(* CODESYS project BODAS-HelloWorld

Project tree, tasks and I/O mapping:
  BODAS_RC18_12_40 : BODAS_RC18-12_27-18_40, Bosch Rexroth AG, version 3.5.21.0
    application Application
      libraries: BODAS_RC18-12_27-18_40, 3.0.1 (Bosch Rexroth AG); BODAS_RC18-12_27-18_40-DST, 2.3.0 (Bosch Rexroth AG); BODAS_RC18-12_27-18_40-PR4, 2.3.0 (Bosch Rexroth AG); Util, 3.5.19.0 (System)
      task Os10msProc (cyclic, interval 10 ms, priority 1) calls MAIN_TASK_PRG
      00 Init/
        FunctionBlocks/
        program INIT_PRG [ST]: INIT_cfgInputs, INIT_cfgOutputs, INIT_initCAN, INIT_initNVM, INIT_initSys, INIT_initUDS
        Programs/
      01 MainTask/
        00 Startlock/
          FunctionBlocks/
          Programs/
        01 Inputs/
          FunctionBlocks/
          program PRG_Inputs [ST]: ACT_InitInputs
          Programs/
        02 Outputs/
          FunctionBlocks/
          program PRG_Outputs [ST]: ACT_HandleInhibit, ACT_InitOutputs
          program PRG_SafeOuts [ST]: ACT_InitSafeOutputs
          Programs/
        03 Communication/
          00 CAN/
            Function/
            FunctionBlocks/
            program PRG_CANIn [ST]
            program PRG_CANOut [ST]
            Programs/
          01 ISOBUSJ1939/
            FunctionBlocks/
            program PRG_ISOBUSJ1939 [ST]
            Programs/
          02 CANopen/
        04 Hydraulics/
          FunctionBlocks/
          Programs/
        05 Engine/
          FunctionBlocks/
          Programs/
        06 Drivetrain/
          FunctionBlocks/
          Programs/
        07 HMI/
          FunctionBlocks/
          Programs/
        10 Service/
          FunctionBlocks/
          program PRG_UDS [ST]: ACT_InitUDS
          Programs/
            program UDS_DefaultCallback [ST]
            function UDS_Diag_ChkLvl [ST]
            function UDS_ReadCallback [ST]
            program UDS_RoutineCallback [ST]
            function UDS_WriteCallback [ST]
        11 Parameters/
          FunctionBlocks/
          Functions/
            function FUNC_DbgMgrRisingEdgeDetn [ST]
          program PRG_DebugManager [ST]: ACT_InitDebugManager
          Programs/
            program PRG_NVMConfig [ST]
        20_Errors/
          FunctionBlocks/
          Functions/
          program PRG_ErrMemMgr [ST]: ACT_ClrDFESEntry, ACT_GetDFESEntry
          program PRG_HandleErrors [ST]: ACT_InitHandleErrors
          Programs/
      02 EasyConfig/
        DSM_easyConfig/
          GVL/
            global variables GVL_debounceMethod
          Structure/
            data type DFC_bds_NoDeb0x8000
            data type DFC_bds_NoDeb0x8001
            data type DFC_bds_NoDeb0x8002
            data type DFC_bds_NoDeb0x8003
            data type DFC_bds_NoDeb0x8004
            data type DFC_bds_NoDeb0x8005
            data type DFC_bds_NoDeb0x8006
            data type DFC_bds_NoDeb0x8007
            data type DFC_bds_NoDeb0x8008
            data type DFC_bds_NoDeb0x8009
            data type DFC_bds_NoDeb0x800a
            data type DFC_bds_NoDeb0x800b
            data type DFC_bds_NoDeb0x800c
            data type DFC_bds_NoDeb0x800d
            data type DFC_bds_NoDeb0x800e
            data type DFC_bds_NoDeb0x800f
            data type DFC_bds_NoDeb0x8010
            data type DFC_bds_NoDeb0x8011
            data type DFC_bds_NoDeb0x8012
            data type DFC_bds_NoDeb0x8013
            data type DFC_bds_NoDeb0x8014
            data type DFC_bds_NoDeb0x8015
            data type DFC_bds_NoDeb0x8016
            data type DFC_bds_NoDeb0x8017
            data type DFC_bds_NoDeb0x8018
            data type DFC_bds_NoDeb0x8019
            data type DFC_bds_NoDeb0x801a
            data type DFC_bds_NoDeb0x801b
            data type DFC_bds_NoDeb0x801c
            data type DFC_bds_NoDeb0x801d
            data type DFC_bds_NoDeb0x801e
            data type DFC_bds_NoDeb0x801f
            data type DFC_bds_NoDeb0x8020
            data type DFC_bds_NoDeb0x8021
            data type DFC_bds_NoDeb0x8022
            data type DFC_bds_NoDeb0x8023
            data type DFC_bds_NoDeb0x8024
            data type DFC_bds_NoDeb0x8025
            data type DFC_bds_NoDeb0x8026
            data type DFC_bds_NoDeb0x8027
            data type DFC_bds_NoDeb0x8028
            data type DFC_bds_NoDeb0x8029
            data type DFC_bds_NoDeb0x802a
            data type DFC_bds_NoDeb0x802b
            data type DFC_bds_NoDeb0x802c
            data type DFC_bds_NoDeb0x802d
            data type DFC_bds_NoDeb0x802e
            data type DFC_bds_NoDeb0x802f
            data type DFC_bds_NoDeb0x8030
            data type DFC_bds_NoDeb0x8031
            data type DFC_bds_NoDeb0x8032
            data type DFC_bds_NoDeb0x8033
            data type DFC_bds_NoDeb0x8034
            data type DFC_bds_NoDeb0x8035
            data type DFC_bds_NoDeb0x8036
            data type DFC_bds_NoDeb0x8037
            data type DFC_bds_NoDeb0x8038
            data type DFC_bds_NoDeb0x8039
            data type DFC_bds_NoDeb0x803a
            data type DFC_bds_NoDeb0x803b
            data type DFC_bds_NoDeb0x803c
            data type DFC_bds_NoDeb0x803d
            data type DFC_bds_NoDeb0x803e
            data type DFC_bds_NoDeb0x803f
            data type DFC_bds_NoDeb0x8040
            data type DFC_bds_NoDeb0x8041
            data type DFC_bds_NoDeb0x8042
            data type DFC_bds_NoDeb0x8043
            data type DFC_bds_NoDeb0x8044
            data type DFC_bds_NoDeb0x8045
            data type DFC_bds_NoDeb0x8046
            data type DFC_bds_NoDeb0x8047
            data type DFC_bds_NoDeb0x8048
            data type DFC_bds_NoDeb0x8049
            data type DFC_bds_NoDeb0x804a
            data type DFC_bds_NoDeb0x804b
            data type DFC_bds_NoDeb0x804c
            data type DFC_bds_NoDeb0x804d
            data type DFC_bds_NoDeb0x804e
            data type DFC_bds_NoDeb0x804f
            data type DFC_bds_NoDeb0x8050
            data type DFC_bds_NoDeb0x8051
            data type DFC_bds_NoDeb0x8052
            data type DFC_bds_NoDeb0x8053
            data type DFC_bds_NoDeb0x8054
            data type DFC_bds_NoDeb0x8055
            data type DFC_bds_NoDeb0x8056
            data type DFC_bds_NoDeb0x8057
            data type DFC_bds_NoDeb0x8058
            data type DFC_bds_NoDeb0x8059
            data type DFC_bds_NoDeb0x805a
            data type DFC_bds_NoDeb0x805b
            data type DFC_bds_NoDeb0x805c
            data type DFC_bds_NoDeb0x805d
            data type DFC_bds_NoDeb0x805e
            data type DFC_bds_NoDeb0x805f
            data type DFC_bds_NoDeb0x8060
            data type DFC_bds_NoDeb0x8061
            data type DFC_bds_NoDeb0x8062
            data type DFC_bds_NoDeb0x8063
            data type DFC_bds_NoDeb0x8064
            data type DFC_bds_NoDeb0x8065
            data type DFC_bds_NoDeb0x8066
            data type DFC_bds_NoDeb0x8067
            data type DFC_bds_NoDeb0x8068
            data type DFC_bds_NoDeb0x8069
            data type DFC_bds_NoDeb0x806a
            data type DFC_bds_NoDeb0x806b
            data type DFC_bds_NoDeb0x806c
            data type DFC_bds_NoDeb0x806d
            data type DFC_bds_NoDeb0x806e
            data type DFC_bds_NoDeb0x806f
            data type DFC_bds_NoDeb0x8070
            data type DFC_bds_NoDeb0x8071
            data type DFC_bds_NoDeb0x8072
            data type DFC_bds_NoDeb0x8073
            data type DFC_bds_NoDeb0x8074
            data type DFC_bds_NoDeb0x8075
            data type DFC_bds_NoDeb0x8076
            data type DFC_bds_NoDeb0x8077
            data type DFC_bds_NoDeb0x8078
            data type DFC_bds_NoDeb0x8079
            data type DFC_bds_NoDeb0x807a
            data type DFC_bds_NoDeb0x807b
            data type DFC_bds_NoDeb0x807c
            data type DFC_bds_NoDeb0x807d
            data type DFC_bds_NoDeb0x807e
            data type DFC_bds_NoDeb0x807f
            data type DFC_bds_NoDeb0x8080
            data type DFC_bds_NoDeb0x8081
            data type DFC_bds_NoDeb0x8082
            data type DFC_bds_NoDeb0x8083
            data type DFC_bds_NoDeb0x8084
            data type DFC_bds_NoDeb0x8085
            data type DFC_bds_NoDeb0x8086
            data type DFC_bds_NoDeb0x8087
            data type DFC_bds_NoDeb0x8088
            data type DFC_bds_NoDeb0x8089
            data type DFC_bds_NoDeb0x808a
            data type DFC_bds_NoDeb0x808b
            data type DFC_bds_NoDeb0x808c
            data type DFC_bds_NoDeb0x808d
            data type DFC_bds_NoDeb0x808e
            data type DFC_bds_NoDeb0x808f
            data type DFC_bds_NoDeb0x8090
            data type DFC_bds_NoDeb0x8091
            data type DFC_bds_NoDeb0x8092
            data type DFC_bds_NoDeb0x8093
            data type DFC_bds_NoDeb0x8094
            data type DFC_bds_NoDeb0x8095
            data type DFC_bds_NoDeb0x8096
            data type DFC_bds_NoDeb0x8097
            data type DFC_bds_NoDeb0x8098
            data type DFC_bds_NoDeb0x8099
            data type DFC_bds_NoDeb0x809a
            data type DFC_bds_NoDeb0x809b
            data type DFC_bds_NoDeb0x809c
            data type DFC_bds_NoDeb0x809d
            data type DFC_bds_NoDeb0x809e
            data type DFC_bds_NoDeb0x809f
            data type DFC_bds_NoDeb0x80a0
            data type DFC_bds_NoDeb0x80a1
            data type DFC_bds_NoDeb0x80a2
            data type DFC_bds_NoDeb0x80a3
            data type DFC_bds_NoDeb0x80a4
            data type DFC_bds_NoDeb0x80a5
            data type DFC_bds_NoDeb0x80a6
            data type DFC_bds_NoDeb0x80a7
            data type DFC_bds_NoDeb0x80a8
            data type DFC_bds_NoDeb0x80a9
            data type DFC_bds_NoDeb0x80aa
            data type DFC_bds_NoDeb0x80ab
            data type DFC_bds_NoDeb0x80ac
            data type DFC_bds_NoDeb0x80ad
            data type DFC_bds_NoDeb0x80ae
            data type DFC_bds_NoDeb0x80af
            data type DFC_bds_NoDeb0x80b0
            data type DFC_bds_NoDeb0x80b1
            data type DFC_bds_NoDeb0x80b2
            data type DFC_bds_NoDeb0x80b3
            data type DFC_bds_NoDeb0x80b4
            data type DFC_bds_NoDeb0x80b5
            data type DFC_bds_NoDeb0x80b6
            data type DFC_bds_NoDeb0x80b7
            data type DFC_bds_NoDeb0x80b8
            data type DFC_bds_NoDeb0x80b9
            data type DFC_bds_NoDeb0x80ba
            data type DFC_bds_NoDeb0x80bb
            data type DFC_bds_NoDeb0x80bc
            data type DFC_bds_NoDeb0x80bd
            data type DFC_bds_NoDeb0x80be
            data type DFC_bds_NoDeb0x80bf
            data type DFC_bds_NoDeb0x80c0
            data type DFC_bds_NoDeb0x80c1
            data type DFC_bds_NoDeb0x80c2
            data type DFC_bds_NoDeb0x80c3
            data type DFC_bds_NoDeb0x80c4
            data type DFC_bds_NoDeb0x80c5
            data type DFC_bds_NoDeb0x80c6
            data type DFC_bds_NoDeb0x80c7
            data type DFC_bds_NoDeb0x80c8
            data type DFC_bds_NoDeb0x80c9
            data type DFC_bds_NoDeb0x80ca
            data type DFC_bds_NoDeb0x80cb
            data type DFC_bds_NoDeb0x80cc
            data type DFC_bds_NoDeb0x80cd
            data type DFC_bds_NoDeb0x80ce
            data type DFC_bds_NoDeb0x80cf
            data type DFC_bds_NoDeb0x80d0
            data type DFC_bds_NoDeb0x80d1
            data type DFC_bds_NoDeb0x80d2
            data type DFC_bds_NoDeb0x80d3
            data type DFC_bds_NoDeb0x80d4
            data type DFC_bds_NoDeb0x80d5
            data type DFC_bds_NoDeb0x80d6
            data type DFC_bds_NoDeb0x80d7
            data type DFC_bds_NoDeb0x80d8
            data type DFC_bds_NoDeb0x80d9
            data type DFC_bds_NoDeb0x80da
            data type DFC_bds_NoDeb0x80db
            data type DFC_bds_NoDeb0x80dc
            data type DFC_bds_NoDeb0x80dd
            data type DFC_bds_NoDeb0x80de
            data type DFC_bds_NoDeb0x80df
            data type DFC_bds_NoDeb0x80e0
            data type DFC_bds_NoDeb0x80e1
            data type DFC_bds_NoDeb0x80e2
            data type DFC_bds_NoDeb0x80e3
            data type DFC_bds_NoDeb0x80e4
            data type DFC_bds_NoDeb0x80e5
            data type DFC_bds_NoDeb0x80e6
            data type DFC_bds_NoDeb0x80e7
            data type DFC_bds_NoDeb0x80e8
            data type DFC_bds_NoDeb0x80e9
            data type DFC_bds_NoDeb0x80ea
            data type DFC_bds_NoDeb0x80eb
            data type DFC_bds_NoDeb0x80ec
            data type DFC_bds_NoDeb0x80ed
            data type DFC_bds_NoDeb0x80ee
            data type DFC_bds_NoDeb0x80ef
            data type DFC_bds_NoDeb0x80f0
            data type DFC_bds_NoDeb0x80f1
            data type DFC_bds_NoDeb0x80f2
            data type DFC_bds_NoDeb0x80f3
            data type DFC_bds_NoDeb0x80f4
            data type DFC_bds_NoDeb0x80f5
            data type DFC_bds_NoDeb0x80f6
            data type DFC_bds_NoDeb0x80f7
            data type DFC_bds_NoDeb0x80f8
            data type DFC_bds_NoDeb0x80f9
            data type DFC_bds_NoDeb0x80fa
            data type DFC_bds_NoDeb0x80fb
            data type DFC_bds_NoDeb0x80fc
            data type DFC_bds_NoDeb0x80fd
            data type DFC_bds_NoDeb0x80fe
            data type DFC_bds_NoDeb0x80ff
            data type DFC_bds_NoDeb0x8100
            data type DFC_bds_NoDeb0x8101
            data type DFC_bds_NoDeb0x8102
            data type DFC_bds_NoDeb0x8103
            data type DFC_bds_NoDeb0x8104
            data type DFC_bds_NoDeb0x8105
            data type DFC_bds_NoDeb0x8106
            data type DFC_bds_NoDeb0x8107
            data type DFC_bds_NoDeb0x8108
            data type DFC_bds_NoDeb0x8109
            data type DFC_bds_NoDeb0x810a
            data type DFC_bds_NoDeb0x810b
            data type DFC_bds_NoDeb0x810c
            data type DFC_bds_NoDeb0x810d
            data type DFC_bds_NoDeb0x810e
            data type DFC_bds_NoDeb0x810f
            data type DFC_bds_NoDeb0x8110
            data type DFC_bds_NoDeb0x8111
            data type DFC_bds_NoDeb0x8112
            data type DFC_bds_NoDeb0x8113
            data type DFC_bds_NoDeb0x8114
            data type DFC_bds_NoDeb0x8115
            data type DFC_bds_NoDeb0x8116
            data type DFC_bds_NoDeb0x8117
            data type DFC_bds_NoDeb0x8118
            data type DFC_bds_NoDeb0x8119
            data type DFC_bds_NoDeb0x811a
            data type DFC_bds_NoDeb0x811b
            data type DFC_bds_NoDeb0x811c
            data type DFC_bds_NoDeb0x811d
            data type DFC_bds_NoDeb0x811e
            data type DFC_bds_NoDeb0x811f
            data type DFC_bds_NoDeb0x8120
            data type DFC_bds_NoDeb0x8121
            data type DFC_bds_NoDeb0x8122
            data type DFC_bds_NoDeb0x8123
            data type DFC_bds_NoDeb0x8124
            data type DFC_bds_NoDeb0x8125
            data type DFC_bds_NoDeb0x8126
            data type DFC_bds_NoDeb0x8127
            data type DFC_bds_NoDeb0x8128
            data type DFC_bds_NoDeb0x8129
            data type DFC_bds_NoDeb0x812a
            data type DFC_bds_NoDeb0x8C01
            data type DFC_bds_NoDeb0x8C02
            data type DFC_bds_NoDeb0x8C03
            data type DFC_bds_TiInRow0x8B01
            data type DFC_bds_TiInRow0x8B02
            data type DFC_bds_TiInRow0x8B03
            data type DFC_bds_TiUpDwn0x8A01
            data type DFC_bds_TiUpDwn0x8A02
            data type DFC_bds_TiUpDwn0x8A03
            data type DFC_CAN_E_TIMEOUT
            data type DFC_CANSM_E_BUS_OFF_NETWORK_0
            data type DFC_CANSM_E_BUS_OFF_NETWORK_1
            data type DFC_CANSM_E_BUS_OFF_NETWORK_2
            data type DFC_CANSM_E_BUS_OFF_NETWORK_3
            data type DFC_CANTRCV_E_NO_TRCV_CONTROL_0
            data type DFC_Com_numWhlIncFrtLeft
            data type DFC_Com_stWhlSensRrRht
            data type DFC_Com_trqClthTCSDCSDes
            data type DFC_Com_vWhlRrL
            data type DFC_ComChksACC_06
            data type DFC_ComChksBMS_01
            data type DFC_ComChksESP_02
            data type DFC_ComChksESP_05
            data type DFC_ComChksESP_07
            data type DFC_ComChksESP_10
            data type DFC_ComChksESP_19
            data type DFC_ComChksESP_20
            data type DFC_ComChksESP_21
            data type DFC_ComChksKlemmen_Status_01
            data type DFC_ComCntACC_06
            data type DFC_ComCntBMS_01
            data type DFC_ComCntESP_02
            data type DFC_ComCntESP_05
            data type DFC_ComCntESP_07
            data type DFC_ComCntESP_10
            data type DFC_ComCntESP_19
            data type DFC_ComCntESP_20
            data type DFC_ComCntESP_21
            data type DFC_ComCntKlemmen_Status_01
            data type DFC_ComDlcACC_06
            data type DFC_ComDlcESP_02
            data type DFC_ComDlcESP_05
            data type DFC_ComDlcESP_07
            data type DFC_ComDlcESP_10
            data type DFC_ComDlcESP_19
            data type DFC_ComDlcESP_20
            data type DFC_ComDlcESP_21
            data type DFC_COMM_E_NET_START_IND_CHANNEL_0
            data type DFC_COMM_E_NET_START_IND_CHANNEL_1
            data type DFC_COMM_E_NET_START_IND_CHANNEL_2
            data type DFC_COMM_E_NET_START_IND_CHANNEL_3
            data type DFC_COMM_E_NET_START_IND_CHANNEL_4
            data type DFC_COMM_E_NET_START_IND_CHANNEL_5
            data type DFC_ComTOutACC_06
            data type DFC_ComTOutESP_02
            data type DFC_ComTOutESP_05
            data type DFC_ComTOutESP_07
            data type DFC_ComTOutESP_10
            data type DFC_ComTOutESP_19
            data type DFC_ComTOutESP_20
            data type DFC_ComTOutESP_21
            data type DFC_DevLibBattUHi
            data type DFC_DevLibBattULo
            data type DFC_DSMDummy
            data type DFC_LIN_E_TIMEOUT
            data type DFC_MoCSOPICO
            data type DFC_MoFVarPostBldSel
            data type DFC_MoSysCtrlReIni
            data type DFC_MOXEMM_SMU_ALM0_0
            data type DFC_MOXEMM_SMU_ALM0_10
            data type DFC_MOXEMM_SMU_ALM0_11
            data type DFC_MOXEMM_SMU_ALM0_13
            data type DFC_MOXEMM_SMU_ALM0_14
            data type DFC_MOXEMM_SMU_ALM0_1
            data type DFC_MOXEMM_SMU_ALM0_22
            data type DFC_MOXEMM_SMU_ALM0_23
            data type DFC_MOXEMM_SMU_ALM0_2
            data type DFC_MOXEMM_SMU_ALM0_4
            data type DFC_MOXEMM_SMU_ALM0_5
            data type DFC_MOXEMM_SMU_ALM0_7
            data type DFC_MOXEMM_SMU_ALM0_8
            data type DFC_MOXEMM_SMU_ALM10_16
            data type DFC_MOXEMM_SMU_ALM10_17
            data type DFC_MOXEMM_SMU_ALM10_21
            data type DFC_MOXEMM_SMU_ALM11_0
            data type DFC_MOXEMM_SMU_ALM11_1
            data type DFC_MOXEMM_SMU_ALM11_2
            data type DFC_MOXEMM_SMU_ALM11_3
            data type DFC_MOXEMM_SMU_ALM11_4
            data type DFC_MOXEMM_SMU_ALM11_5
            data type DFC_MOXEMM_SMU_ALM11_8
            data type DFC_MOXEMM_SMU_ALM11_9
            data type DFC_MOXEMM_SMU_ALM1_0
            data type DFC_MOXEMM_SMU_ALM1_10
            data type DFC_MOXEMM_SMU_ALM1_11
            data type DFC_MOXEMM_SMU_ALM1_13
            data type DFC_MOXEMM_SMU_ALM1_14
            data type DFC_MOXEMM_SMU_ALM1_1
            data type DFC_MOXEMM_SMU_ALM1_22
            data type DFC_MOXEMM_SMU_ALM1_23
            data type DFC_MOXEMM_SMU_ALM1_2
            data type DFC_MOXEMM_SMU_ALM1_4
            data type DFC_MOXEMM_SMU_ALM1_5
            data type DFC_MOXEMM_SMU_ALM1_7
            data type DFC_MOXEMM_SMU_ALM1_8
            data type DFC_MOXEMM_SMU_ALM21_0
            data type DFC_MOXEMM_SMU_ALM21_16
            data type DFC_MOXEMM_SMU_ALM21_3
            data type DFC_MOXEMM_SMU_ALM2_10
            data type DFC_MOXEMM_SMU_ALM2_11
            data type DFC_MOXEMM_SMU_ALM2_13
            data type DFC_MOXEMM_SMU_ALM2_14
            data type DFC_MOXEMM_SMU_ALM2_1
            data type DFC_MOXEMM_SMU_ALM2_22
            data type DFC_MOXEMM_SMU_ALM2_23
            data type DFC_MOXEMM_SMU_ALM2_2
            data type DFC_MOXEMM_SMU_ALM2_4
            data type DFC_MOXEMM_SMU_ALM2_5
            data type DFC_MOXEMM_SMU_ALM2_7
            data type DFC_MOXEMM_SMU_ALM2_8
            data type DFC_MOXEMM_SMU_ALM3_10
            data type DFC_MOXEMM_SMU_ALM3_11
            data type DFC_MOXEMM_SMU_ALM3_13
            data type DFC_MOXEMM_SMU_ALM3_14
            data type DFC_MOXEMM_SMU_ALM3_1
            data type DFC_MOXEMM_SMU_ALM3_22
            data type DFC_MOXEMM_SMU_ALM3_23
            data type DFC_MOXEMM_SMU_ALM3_2
            data type DFC_MOXEMM_SMU_ALM3_4
            data type DFC_MOXEMM_SMU_ALM3_5
            data type DFC_MOXEMM_SMU_ALM3_7
            data type DFC_MOXEMM_SMU_ALM3_8
            data type DFC_MOXEMM_SMU_ALM6_0
            data type DFC_MOXEMM_SMU_ALM6_11
            data type DFC_MOXEMM_SMU_ALM6_12
            data type DFC_MOXEMM_SMU_ALM6_14
            data type DFC_MOXEMM_SMU_ALM6_15
            data type DFC_MOXEMM_SMU_ALM6_17
            data type DFC_MOXEMM_SMU_ALM6_18
            data type DFC_MOXEMM_SMU_ALM6_20
            data type DFC_MOXEMM_SMU_ALM6_21
            data type DFC_MOXEMM_SMU_ALM6_25
            data type DFC_MOXEMM_SMU_ALM6_2
            data type DFC_MOXEMM_SMU_ALM6_4
            data type DFC_MOXEMM_SMU_ALM6_5
            data type DFC_MOXEMM_SMU_ALM6_7
            data type DFC_MOXEMM_SMU_ALM6_8
            data type DFC_MOXEMM_SMU_ALM7_12
            data type DFC_MOXEMM_SMU_ALM7_13
            data type DFC_MOXEMM_SMU_ALM7_14
            data type DFC_MOXEMM_SMU_ALM7_15
            data type DFC_MOXEMM_SMU_ALM7_16
            data type DFC_MOXEMM_SMU_ALM7_17
            data type DFC_MOXEMM_SMU_ALM7_1
            data type DFC_MOXEMM_SMU_ALM7_20
            data type DFC_MOXEMM_SMU_ALM7_25
            data type DFC_MOXEMM_SMU_ALM7_26
            data type DFC_MOXEMM_SMU_ALM7_28
            data type DFC_MOXEMM_SMU_ALM7_29
            data type DFC_MOXEMM_SMU_ALM7_2
            data type DFC_MOXEMM_SMU_ALM7_30
            data type DFC_MOXEMM_SMU_ALM7_31
            data type DFC_MOXEMM_SMU_ALM8_0
            data type DFC_MOXEMM_SMU_ALM8_10
            data type DFC_MOXEMM_SMU_ALM8_11
            data type DFC_MOXEMM_SMU_ALM8_12
            data type DFC_MOXEMM_SMU_ALM8_13
            data type DFC_MOXEMM_SMU_ALM8_16
            data type DFC_MOXEMM_SMU_ALM8_18
            data type DFC_MOXEMM_SMU_ALM8_1
            data type DFC_MOXEMM_SMU_ALM8_2
            data type DFC_MOXEMM_SMU_ALM8_30
            data type DFC_MOXEMM_SMU_ALM8_31
            data type DFC_MOXEMM_SMU_ALM8_3
            data type DFC_MOXEMM_SMU_ALM8_4
            data type DFC_MOXEMM_SMU_ALM9_0
            data type DFC_MOXEMM_SMU_ALM9_15
            data type DFC_MOXEMM_SMU_ALM9_1
            data type DFC_MOXEMM_SMU_ALM9_3
            data type DFC_MoXEMMHwLTLBIST
            data type DFC_MoXEMMHwLTMBIST
            data type DFC_MoXEMMHwLTMCUFW
            data type DFC_MoXEMMHwLTMonBIST
            data type DFC_MoXEMMHwLTRegMonTest
            data type DFC_MoXEMMHwLTStbySMUAlvTest
        easyConfig_import/
          BDL/
          bds_in_ec/
          bds_in_legacy_ec/
          bds_out_ec/
          bds_sent_ec/
          bds_sysIo_ec/
          bds_sysPb_ec/
        Lin_CanSignals_easyConfig/
          global variables GVL_linCanSignals_easyConfig
      03 PrivateLibrary/
        DataTypes/
          DebugManager/
          ErrMemMgr/
          ISOBUSJ1939/
          MainTask/
      global variables GlobalVariables
      program MAIN_TASK_PRG [ST]: CAN_OUT, ERRORS, INIT, INPUTS, OUTPUTS, POSTRUN, READ_PARAMETERS, RUN, STARTLOCK
*)

// BODAS_RC18_12_40/Application/02 EasyConfig/DSM_easyConfig/Structure/DFC_bds_NoDeb0x8000
{attribute 'external_name' := 'cmp_rts_DFC_bds_NoDeb0x8000'}
TYPE DFC_bds_NoDeb0x8000 : STRUCT
        DTC            : UDINT := 16#800000;
        DFCid          : UINT  := 721;
        debounceMethod : USINT := NO_DEBOUNCE;
    END_STRUCT
END_TYPE

// BODAS_RC18_12_40/Application/02 EasyConfig/DSM_easyConfig/Structure/DFC_bds_NoDeb0x8001
{attribute 'external_name' := 'cmp_rts_DFC_bds_NoDeb0x8001'}
TYPE DFC_bds_NoDeb0x8001 : STRUCT
        DTC            : UDINT := 16#800100;
        DFCid          : UINT  := 722;
        debounceMethod : USINT := NO_DEBOUNCE;
    END_STRUCT
END_TYPE

// BODAS_RC18_12_40/Application/02 EasyConfig/DSM_easyConfig/Structure/DFC_bds_NoDeb0x8002
{attribute 'external_name' := 'cmp_rts_DFC_bds_NoDeb0x8002'}
TYPE DFC_bds_NoDeb0x8002 : STRUCT
        DTC            : UDINT := 16#800200;
        DFCid          : UINT  := 723;
        debounceMethod : USINT := NO_DEBOUNCE;
    END_STRUCT
END_TYPE

// BODAS_RC18_12_40/Application/02 EasyConfig/DSM_easyConfig/Structure/DFC_bds_NoDeb0x8003
{attribute 'external_name' := 'cmp_rts_DFC_bds_NoDeb0x8003'}
TYPE DFC_bds_NoDeb0x8003 : STRUCT
        DTC            : UDINT := 16#800300;
        DFCid          : UINT  := 724;
        debounceMethod : USINT := NO_DEBOUNCE;
    END_STRUCT
END_TYPE

// BODAS_RC18_12_40/Application/02 EasyConfig/DSM_easyConfig/Structure/DFC_bds_NoDeb0x8004
{attribute 'external_name' := 'cmp_rts_DFC_bds_NoDeb0x8004'}
TYPE DFC_bds_NoDeb0x8004 : STRUCT
        DTC            : UDINT := 16#800400;
        DFCid          : UINT  := 725;
        debounceMethod : USINT := NO_DEBOUNCE;
    END_STRUCT
END_TYPE

// BODAS_RC18_12_40/Application/02 EasyConfig/DSM_easyConfig/Structure/DFC_bds_NoDeb0x8005
{attribute 'external_name' := 'cmp_rts_DFC_bds_NoDeb0x8005'}
TYPE DFC_bds_NoDeb0x8005 :
STRUCT
	DTC: UDINT := 16#800500;
	DFCid: UINT := 726;
	debounceMethod: USINT := NO_DEBOUNCE;
END_STRUCT
END_TYPE

// BODAS_RC18_12_40/Application/02 EasyConfig/DSM_easyConfig/Structure/DFC_bds_NoDeb0x8006
{attribute 'external_name' := 'cmp_rts_DFC_bds_NoDeb0x8006'}
TYPE DFC_bds_NoDeb0x8006 : STRUCT
        DTC            : UDINT := 16#800600;
        DFCid          : UINT  := 727;
        debounceMethod : USINT := NO_DEBOUNCE;
    END_STRUCT
END_TYPE

// BODAS_RC18_12_40/Application/02 EasyConfig/DSM_easyConfig/Structure/DFC_bds_NoDeb0x8007
{attribute 'external_name' := 'cmp_rts_DFC_bds_NoDeb0x8007'}
TYPE DFC_bds_NoDeb0x8007 : STRUCT
        DTC            : UDINT := 16#800700;
        DFCid          : UINT  := 728;
        debounceMethod : USINT := NO_DEBOUNCE;
    END_STRUCT
END_TYPE

// BODAS_RC18_12_40/Application/02 EasyConfig/DSM_easyConfig/Structure/DFC_bds_NoDeb0x8008
{attribute 'external_name' := 'cmp_rts_DFC_bds_NoDeb0x8008'}
TYPE DFC_bds_NoDeb0x8008 : STRUCT
        DTC            : UDINT := 16#800800;
        DFCid          : UINT  := 729;
        debounceMethod : USINT := NO_DEBOUNCE;
    END_STRUCT
END_TYPE

// BODAS_RC18_12_40/Application/02 EasyConfig/DSM_easyConfig/Structure/DFC_bds_NoDeb0x8009
{attribute 'external_name' := 'cmp_rts_DFC_bds_NoDeb0x8009'}
TYPE DFC_bds_NoDeb0x8009 :
STRUCT
	DTC: UDINT := 16#800900;
	DFCid: UINT := 730;
	debounceMethod: USINT := NO_DEBOUNCE;
END_STRUCT
END_TYPE

// BODAS_RC18_12_40/Application/02 EasyConfig/DSM_easyConfig/Structure/DFC_bds_NoDeb0x800a
{attribute 'external_name' := 'cmp_rts_DFC_bds_NoDeb0x800a'}
TYPE DFC_bds_NoDeb0x800a : STRUCT
        DTC            : UDINT := 16#800A00;
        DFCid          : UINT  := 731;
        debounceMethod : USINT := NO_DEBOUNCE;
    END_STRUCT
END_TYPE

// BODAS_RC18_12_40/Application/02 EasyConfig/DSM_easyConfig/Structure/DFC_bds_NoDeb0x800b
{attribute 'external_name' := 'cmp_rts_DFC_bds_NoDeb0x800b'}
TYPE DFC_bds_NoDeb0x800b : STRUCT
        DTC            : UDINT := 16#800B00;
        DFCid          : UINT  := 732;
        debounceMethod : USINT := NO_DEBOUNCE;
    END_STRUCT
END_TYPE

// BODAS_RC18_12_40/Application/02 EasyConfig/DSM_easyConfig/Structure/DFC_bds_NoDeb0x800c
{attribute 'external_name' := 'cmp_rts_DFC_bds_NoDeb0x800c'}
TYPE DFC_bds_NoDeb0x800c :
STRUCT
	DTC: UDINT := 16#800C00;
	DFCid: UINT := 733;
	debounceMethod: USINT := NO_DEBOUNCE;
END_STRUCT
END_TYPE

// BODAS_RC18_12_40/Application/02 EasyConfig/DSM_easyConfig/Structure/DFC_bds_NoDeb0x800d
{attribute 'external_name' := 'cmp_rts_DFC_bds_NoDeb0x800d'}
TYPE DFC_bds_NoDeb0x800d : STRUCT
        DTC            : UDINT := 16#800D00;
        DFCid          : UINT  := 734;
        debounceMethod : USINT := NO_DEBOUNCE;
    END_STRUCT
END_TYPE

// BODAS_RC18_12_40/Application/02 EasyConfig/DSM_easyConfig/Structure/DFC_bds_NoDeb0x800e
{attribute 'external_name' := 'cmp_rts_DFC_bds_NoDeb0x800e'}
TYPE DFC_bds_NoDeb0x800e :
STRUCT
	DTC: UDINT := 16#800E00;
	DFCid: UINT := 735;
	debounceMethod: USINT := NO_DEBOUNCE;
END_STRUCT
END_TYPE

// BODAS_RC18_12_40/Application/02 EasyConfig/DSM_easyConfig/Structure/DFC_bds_NoDeb0x800f
{attribute 'external_name' := 'cmp_rts_DFC_bds_NoDeb0x800f'}
TYPE DFC_bds_NoDeb0x800f : STRUCT
        DTC            : UDINT := 16#800F00;
        DFCid          : UINT  := 736;
        debounceMethod : USINT := NO_DEBOUNCE;
    END_STRUCT
END_TYPE

// BODAS_RC18_12_40/Application/02 EasyConfig/DSM_easyConfig/Structure/DFC_bds_NoDeb0x8010
{attribute 'external_name' := 'cmp_rts_DFC_bds_NoDeb0x8010'}
TYPE DFC_bds_NoDeb0x8010 : STRUCT
        DTC            : UDINT := 16#801000;
        DFCid          : UINT  := 737;
        debounceMethod : USINT := NO_DEBOUNCE;
    END_STRUCT
END_TYPE

// BODAS_RC18_12_40/Application/02 EasyConfig/DSM_easyConfig/Structure/DFC_bds_NoDeb0x8011
{attribute 'external_name' := 'cmp_rts_DFC_bds_NoDeb0x8011'}
TYPE DFC_bds_NoDeb0x8011 : STRUCT
        DTC            : UDINT := 16#801100;
        DFCid          : UINT  := 738;
        debounceMethod : USINT := NO_DEBOUNCE;
    END_STRUCT
END_TYPE

// BODAS_RC18_12_40/Application/02 EasyConfig/DSM_easyConfig/Structure/DFC_bds_NoDeb0x8012
{attribute 'external_name' := 'cmp_rts_DFC_bds_NoDeb0x8012'}
TYPE DFC_bds_NoDeb0x8012 : STRUCT
        DTC            : UDINT := 16#801200;
        DFCid          : UINT  := 739;
        debounceMethod : USINT := NO_DEBOUNCE;
    END_STRUCT
END_TYPE

// BODAS_RC18_12_40/Application/02 EasyConfig/DSM_easyConfig/Structure/DFC_bds_NoDeb0x8013
{attribute 'external_name' := 'cmp_rts_DFC_bds_NoDeb0x8013'}
TYPE DFC_bds_NoDeb0x8013 : STRUCT
        DTC            : UDINT := 16#801300;
        DFCid          : UINT  := 740;
        debounceMethod : USINT := NO_DEBOUNCE;
    END_STRUCT
END_TYPE

// BODAS_RC18_12_40/Application/02 EasyConfig/DSM_easyConfig/Structure/DFC_bds_NoDeb0x8014
{attribute 'external_name' := 'cmp_rts_DFC_bds_NoDeb0x8014'}
TYPE DFC_bds_NoDeb0x8014 : STRUCT
        DTC            : UDINT := 16#801400;
        DFCid          : UINT  := 741;
        debounceMethod : USINT := NO_DEBOUNCE;
    END_STRUCT
END_TYPE

// BODAS_RC18_12_40/Application/02 EasyConfig/DSM_easyConfig/Structure/DFC_bds_NoDeb0x8015
{attribute 'external_name' := 'cmp_rts_DFC_bds_NoDeb0x8015'}
TYPE DFC_bds_NoDeb0x8015 : STRUCT
        DTC            : UDINT := 16#801500;
        DFCid          : UINT  := 742;
        debounceMethod : USINT := NO_DEBOUNCE;
    END_STRUCT
END_TYPE

// BODAS_RC18_12_40/Application/02 EasyConfig/DSM_easyConfig/Structure/DFC_bds_NoDeb0x8016
{attribute 'external_name' := 'cmp_rts_DFC_bds_NoDeb0x8016'}
TYPE DFC_bds_NoDeb0x8016 : STRUCT
        DTC            : UDINT := 16#801600;
        DFCid          : UINT  := 743;
        debounceMethod : USINT := NO_DEBOUNCE;
    END_STRUCT
END_TYPE

// BODAS_RC18_12_40/Application/02 EasyConfig/DSM_easyConfig/Structure/DFC_bds_NoDeb0x8017
{attribute 'external_name' := 'cmp_rts_DFC_bds_NoDeb0x8017'}
TYPE DFC_bds_NoDeb0x8017 : STRUCT
        DTC            : UDINT := 16#801700;
        DFCid          : UINT  := 744;
        debounceMethod : USINT := NO_DEBOUNCE;
    END_STRUCT
END_TYPE

// BODAS_RC18_12_40/Application/02 EasyConfig/DSM_easyConfig/Structure/DFC_bds_NoDeb0x8018
{attribute 'external_name' := 'cmp_rts_DFC_bds_NoDeb0x8018'}
TYPE DFC_bds_NoDeb0x8018 : STRUCT
        DTC            : UDINT := 16#801800;
        DFCid          : UINT  := 745;
        debounceMethod : USINT := NO_DEBOUNCE;
    END_STRUCT
END_TYPE

// BODAS_RC18_12_40/Application/02 EasyConfig/DSM_easyConfig/Structure/DFC_bds_NoDeb0x8019
{attribute 'external_name' := 'cmp_rts_DFC_bds_NoDeb0x8019'}
TYPE DFC_bds_NoDeb0x8019 :
STRUCT
	DTC: UDINT := 16#801900;
	DFCid: UINT := 746;
	debounceMethod: USINT := NO_DEBOUNCE;
END_STRUCT
END_TYPE

// BODAS_RC18_12_40/Application/02 EasyConfig/DSM_easyConfig/Structure/DFC_bds_NoDeb0x801a
{attribute 'external_name' := 'cmp_rts_DFC_bds_NoDeb0x801a'}
TYPE DFC_bds_NoDeb0x801a : STRUCT
        DTC            : UDINT := 16#801A00;
        DFCid          : UINT  := 747;
        debounceMethod : USINT := NO_DEBOUNCE;
    END_STRUCT
END_TYPE

// BODAS_RC18_12_40/Application/02 EasyConfig/DSM_easyConfig/Structure/DFC_bds_NoDeb0x801b
{attribute 'external_name' := 'cmp_rts_DFC_bds_NoDeb0x801b'}
TYPE DFC_bds_NoDeb0x801b : STRUCT
        DTC            : UDINT := 16#801B00;
        DFCid          : UINT  := 748;
        debounceMethod : USINT := NO_DEBOUNCE;
    END_STRUCT
END_TYPE

// BODAS_RC18_12_40/Application/02 EasyConfig/DSM_easyConfig/Structure/DFC_bds_NoDeb0x801c
{attribute 'external_name' := 'cmp_rts_DFC_bds_NoDeb0x801c'}
TYPE DFC_bds_NoDeb0x801c :
STRUCT
	DTC: UDINT := 16#801C00;
	DFCid: UINT := 749;
	debounceMethod: USINT := NO_DEBOUNCE;
END_STRUCT
END_TYPE

// BODAS_RC18_12_40/Application/02 EasyConfig/DSM_easyConfig/Structure/DFC_bds_NoDeb0x801d
{attribute 'external_name' := 'cmp_rts_DFC_bds_NoDeb0x801d'}
TYPE DFC_bds_NoDeb0x801d :
STRUCT
	DTC: UDINT := 16#801D00;
	DFCid: UINT := 750;
	debounceMethod: USINT := NO_DEBOUNCE;
END_STRUCT
END_TYPE

// BODAS_RC18_12_40/Application/02 EasyConfig/DSM_easyConfig/Structure/DFC_bds_NoDeb0x801e
{attribute 'external_name' := 'cmp_rts_DFC_bds_NoDeb0x801e'}
TYPE DFC_bds_NoDeb0x801e : STRUCT
        DTC            : UDINT := 16#801E00;
        DFCid          : UINT  := 751;
        debounceMethod : USINT := NO_DEBOUNCE;
    END_STRUCT
END_TYPE

// BODAS_RC18_12_40/Application/02 EasyConfig/DSM_easyConfig/Structure/DFC_bds_NoDeb0x801f
{attribute 'external_name' := 'cmp_rts_DFC_bds_NoDeb0x801f'}
TYPE DFC_bds_NoDeb0x801f : STRUCT
        DTC            : UDINT := 16#801F00;
        DFCid          : UINT  := 752;
        debounceMethod : USINT := NO_DEBOUNCE;
    END_STRUCT
END_TYPE

// BODAS_RC18_12_40/Application/02 EasyConfig/DSM_easyConfig/Structure/DFC_bds_NoDeb0x8020
{attribute 'external_name' := 'cmp_rts_DFC_bds_NoDeb0x8020'}
TYPE DFC_bds_NoDeb0x8020 :
STRUCT
	DTC: UDINT := 16#802000;
	DFCid: UINT := 753;
	debounceMethod: USINT := NO_DEBOUNCE;
END_STRUCT
END_TYPE

// BODAS_RC18_12_40/Application/02 EasyConfig/DSM_easyConfig/Structure/DFC_bds_NoDeb0x8021
{attribute 'external_name' := 'cmp_rts_DFC_bds_NoDeb0x8021'}
TYPE DFC_bds_NoDeb0x8021 : STRUCT
        DTC            : UDINT := 16#802100;
        DFCid          : UINT  := 754;
        debounceMethod : USINT := NO_DEBOUNCE;
    END_STRUCT
END_TYPE

// BODAS_RC18_12_40/Application/02 EasyConfig/DSM_easyConfig/Structure/DFC_bds_NoDeb0x8022
{attribute 'external_name' := 'cmp_rts_DFC_bds_NoDeb0x8022'}
TYPE DFC_bds_NoDeb0x8022 : STRUCT
        DTC            : UDINT := 16#802200;
        DFCid          : UINT  := 755;
        debounceMethod : USINT := NO_DEBOUNCE;
    END_STRUCT
END_TYPE

// BODAS_RC18_12_40/Application/02 EasyConfig/DSM_easyConfig/Structure/DFC_bds_NoDeb0x8023
{attribute 'external_name' := 'cmp_rts_DFC_bds_NoDeb0x8023'}
TYPE DFC_bds_NoDeb0x8023 : STRUCT
        DTC            : UDINT := 16#802300;
        DFCid          : UINT  := 756;
        debounceMethod : USINT := NO_DEBOUNCE;
    END_STRUCT
END_TYPE

// BODAS_RC18_12_40/Application/02 EasyConfig/DSM_easyConfig/Structure/DFC_bds_NoDeb0x8024
{attribute 'external_name' := 'cmp_rts_DFC_bds_NoDeb0x8024'}
TYPE DFC_bds_NoDeb0x8024 : STRUCT
        DTC            : UDINT := 16#802400;
        DFCid          : UINT  := 757;
        debounceMethod : USINT := NO_DEBOUNCE;
    END_STRUCT
END_TYPE

// BODAS_RC18_12_40/Application/02 EasyConfig/DSM_easyConfig/Structure/DFC_bds_NoDeb0x8025
{attribute 'external_name' := 'cmp_rts_DFC_bds_NoDeb0x8025'}
TYPE DFC_bds_NoDeb0x8025 : STRUCT
        DTC            : UDINT := 16#802500;
        DFCid          : UINT  := 758;
        debounceMethod : USINT := NO_DEBOUNCE;
    END_STRUCT
END_TYPE

// BODAS_RC18_12_40/Application/02 EasyConfig/DSM_easyConfig/Structure/DFC_bds_NoDeb0x8026
{attribute 'external_name' := 'cmp_rts_DFC_bds_NoDeb0x8026'}
TYPE DFC_bds_NoDeb0x8026 :
STRUCT
	DTC: UDINT := 16#802600;
	DFCid: UINT := 759;
	debounceMethod: USINT := NO_DEBOUNCE;
END_STRUCT
END_TYPE

// BODAS_RC18_12_40/Application/02 EasyConfig/DSM_easyConfig/Structure/DFC_bds_NoDeb0x8027
{attribute 'external_name' := 'cmp_rts_DFC_bds_NoDeb0x8027'}
TYPE DFC_bds_NoDeb0x8027 : STRUCT
        DTC            : UDINT := 16#802700;
        DFCid          : UINT  := 760;
        debounceMethod : USINT := NO_DEBOUNCE;
    END_STRUCT
END_TYPE

// BODAS_RC18_12_40/Application/02 EasyConfig/DSM_easyConfig/Structure/DFC_bds_NoDeb0x8028
{attribute 'external_name' := 'cmp_rts_DFC_bds_NoDeb0x8028'}
TYPE DFC_bds_NoDeb0x8028 :
STRUCT
	DTC: UDINT := 16#802800;
	DFCid: UINT := 761;
	debounceMethod: USINT := NO_DEBOUNCE;
END_STRUCT
END_TYPE

// BODAS_RC18_12_40/Application/02 EasyConfig/DSM_easyConfig/Structure/DFC_bds_NoDeb0x8029
{attribute 'external_name' := 'cmp_rts_DFC_bds_NoDeb0x8029'}
TYPE DFC_bds_NoDeb0x8029 : STRUCT
        DTC            : UDINT := 16#802900;
        DFCid          : UINT  := 762;
        debounceMethod : USINT := NO_DEBOUNCE;
    END_STRUCT
END_TYPE

// BODAS_RC18_12_40/Application/02 EasyConfig/DSM_easyConfig/Structure/DFC_bds_NoDeb0x802a
{attribute 'external_name' := 'cmp_rts_DFC_bds_NoDeb0x802a'}
TYPE DFC_bds_NoDeb0x802a : STRUCT
        DTC            : UDINT := 16#802A00;
        DFCid          : UINT  := 763;
        debounceMethod : USINT := NO_DEBOUNCE;
    END_STRUCT
END_TYPE

// BODAS_RC18_12_40/Application/02 EasyConfig/DSM_easyConfig/Structure/DFC_bds_NoDeb0x802b
{attribute 'external_name' := 'cmp_rts_DFC_bds_NoDeb0x802b'}
TYPE DFC_bds_NoDeb0x802b : STRUCT
        DTC            : UDINT := 16#802B00;
        DFCid          : UINT  := 764;
        debounceMethod : USINT := NO_DEBOUNCE;
    END_STRUCT
END_TYPE

// BODAS_RC18_12_40/Application/02 EasyConfig/DSM_easyConfig/Structure/DFC_bds_NoDeb0x802c
{attribute 'external_name' := 'cmp_rts_DFC_bds_NoDeb0x802c'}
TYPE DFC_bds_NoDeb0x802c : STRUCT
        DTC            : UDINT := 16#802C00;
        DFCid          : UINT  := 765;
        debounceMethod : USINT := NO_DEBOUNCE;
    END_STRUCT
END_TYPE

// BODAS_RC18_12_40/Application/02 EasyConfig/DSM_easyConfig/Structure/DFC_bds_NoDeb0x802d
{attribute 'external_name' := 'cmp_rts_DFC_bds_NoDeb0x802d'}
TYPE DFC_bds_NoDeb0x802d : STRUCT
        DTC            : UDINT := 16#802D00;
        DFCid          : UINT  := 766;
        debounceMethod : USINT := NO_DEBOUNCE;
    END_STRUCT
END_TYPE

// BODAS_RC18_12_40/Application/02 EasyConfig/DSM_easyConfig/Structure/DFC_bds_NoDeb0x802e
{attribute 'external_name' := 'cmp_rts_DFC_bds_NoDeb0x802e'}
TYPE DFC_bds_NoDeb0x802e : STRUCT
        DTC            : UDINT := 16#802E00;
        DFCid          : UINT  := 767;
        debounceMethod : USINT := NO_DEBOUNCE;
    END_STRUCT
END_TYPE

// BODAS_RC18_12_40/Application/02 EasyConfig/DSM_easyConfig/Structure/DFC_bds_NoDeb0x802f
{attribute 'external_name' := 'cmp_rts_DFC_bds_NoDeb0x802f'}
TYPE DFC_bds_NoDeb0x802f : STRUCT
        DTC            : UDINT := 16#802F00;
        DFCid          : UINT  := 768;
        debounceMethod : USINT := NO_DEBOUNCE;
    END_STRUCT
END_TYPE

// BODAS_RC18_12_40/Application/02 EasyConfig/DSM_easyConfig/Structure/DFC_bds_NoDeb0x8030
{attribute 'external_name' := 'cmp_rts_DFC_bds_NoDeb0x8030'}
TYPE DFC_bds_NoDeb0x8030 : STRUCT
        DTC            : UDINT := 16#803000;
        DFCid          : UINT  := 769;
        debounceMethod : USINT := NO_DEBOUNCE;
    END_STRUCT
END_TYPE

// BODAS_RC18_12_40/Application/02 EasyConfig/DSM_easyConfig/Structure/DFC_bds_NoDeb0x8031
{attribute 'external_name' := 'cmp_rts_DFC_bds_NoDeb0x8031'}
TYPE DFC_bds_NoDeb0x8031 : STRUCT
        DTC            : UDINT := 16#803100;
        DFCid          : UINT  := 770;
        debounceMethod : USINT := NO_DEBOUNCE;
    END_STRUCT
END_TYPE

// BODAS_RC18_12_40/Application/02 EasyConfig/DSM_easyConfig/Structure/DFC_bds_NoDeb0x8032
{attribute 'external_name' := 'cmp_rts_DFC_bds_NoDeb0x8032'}
TYPE DFC_bds_NoDeb0x8032 :
STRUCT
	DTC: UDINT := 16#803200;
	DFCid: UINT := 771;
	debounceMethod: USINT := NO_DEBOUNCE;
END_STRUCT
END_TYPE

// BODAS_RC18_12_40/Application/02 EasyConfig/DSM_easyConfig/Structure/DFC_bds_NoDeb0x8033
{attribute 'external_name' := 'cmp_rts_DFC_bds_NoDeb0x8033'}
TYPE DFC_bds_NoDeb0x8033 : STRUCT
        DTC            : UDINT := 16#803300;
        DFCid          : UINT  := 772;
        debounceMethod : USINT := NO_DEBOUNCE;
    END_STRUCT
END_TYPE

// BODAS_RC18_12_40/Application/02 EasyConfig/DSM_easyConfig/Structure/DFC_bds_NoDeb0x8034
{attribute 'external_name' := 'cmp_rts_DFC_bds_NoDeb0x8034'}
TYPE DFC_bds_NoDeb0x8034 : STRUCT
        DTC            : UDINT := 16#803400;
        DFCid          : UINT  := 773;
        debounceMethod : USINT := NO_DEBOUNCE;
    END_STRUCT
END_TYPE

// BODAS_RC18_12_40/Application/02 EasyConfig/DSM_easyConfig/Structure/DFC_bds_NoDeb0x8035
{attribute 'external_name' := 'cmp_rts_DFC_bds_NoDeb0x8035'}
TYPE DFC_bds_NoDeb0x8035 : STRUCT
        DTC            : UDINT := 16#803500;
        DFCid          : UINT  := 774;
        debounceMethod : USINT := NO_DEBOUNCE;
    END_STRUCT
END_TYPE

// BODAS_RC18_12_40/Application/02 EasyConfig/DSM_easyConfig/Structure/DFC_bds_NoDeb0x8036
{attribute 'external_name' := 'cmp_rts_DFC_bds_NoDeb0x8036'}
TYPE DFC_bds_NoDeb0x8036 : STRUCT
        DTC            : UDINT := 16#803600;
        DFCid          : UINT  := 775;
        debounceMethod : USINT := NO_DEBOUNCE;
    END_STRUCT
END_TYPE

// BODAS_RC18_12_40/Application/02 EasyConfig/DSM_easyConfig/Structure/DFC_bds_NoDeb0x8037
{attribute 'external_name' := 'cmp_rts_DFC_bds_NoDeb0x8037'}
TYPE DFC_bds_NoDeb0x8037 :
STRUCT
	DTC: UDINT := 16#803700;
	DFCid: UINT := 776;
	debounceMethod: USINT := NO_DEBOUNCE;
END_STRUCT
END_TYPE

// BODAS_RC18_12_40/Application/02 EasyConfig/DSM_easyConfig/Structure/DFC_bds_NoDeb0x8038
{attribute 'external_name' := 'cmp_rts_DFC_bds_NoDeb0x8038'}
TYPE DFC_bds_NoDeb0x8038 : STRUCT
        DTC            : UDINT := 16#803800;
        DFCid          : UINT  := 777;
        debounceMethod : USINT := NO_DEBOUNCE;
    END_STRUCT
END_TYPE

// BODAS_RC18_12_40/Application/02 EasyConfig/DSM_easyConfig/Structure/DFC_bds_NoDeb0x8039
{attribute 'external_name' := 'cmp_rts_DFC_bds_NoDeb0x8039'}
TYPE DFC_bds_NoDeb0x8039 : STRUCT
        DTC            : UDINT := 16#803900;
        DFCid          : UINT  := 778;
        debounceMethod : USINT := NO_DEBOUNCE;
    END_STRUCT
END_TYPE

// BODAS_RC18_12_40/Application/02 EasyConfig/DSM_easyConfig/Structure/DFC_bds_NoDeb0x803a
{attribute 'external_name' := 'cmp_rts_DFC_bds_NoDeb0x803a'}
TYPE DFC_bds_NoDeb0x803a :
STRUCT
	DTC: UDINT := 16#803A00;
	DFCid: UINT := 779;
	debounceMethod: USINT := NO_DEBOUNCE;
END_STRUCT
END_TYPE

// BODAS_RC18_12_40/Application/02 EasyConfig/DSM_easyConfig/Structure/DFC_bds_NoDeb0x803b
{attribute 'external_name' := 'cmp_rts_DFC_bds_NoDeb0x803b'}
TYPE DFC_bds_NoDeb0x803b : STRUCT
        DTC            : UDINT := 16#803B00;
        DFCid          : UINT  := 780;
        debounceMethod : USINT := NO_DEBOUNCE;
    END_STRUCT
END_TYPE

// BODAS_RC18_12_40/Application/02 EasyConfig/DSM_easyConfig/Structure/DFC_bds_NoDeb0x803c
{attribute 'external_name' := 'cmp_rts_DFC_bds_NoDeb0x803c'}
TYPE DFC_bds_NoDeb0x803c : STRUCT
        DTC            : UDINT := 16#803C00;
        DFCid          : UINT  := 781;
        debounceMethod : USINT := NO_DEBOUNCE;
    END_STRUCT
END_TYPE

// BODAS_RC18_12_40/Application/02 EasyConfig/DSM_easyConfig/Structure/DFC_bds_NoDeb0x803d
{attribute 'external_name' := 'cmp_rts_DFC_bds_NoDeb0x803d'}
TYPE DFC_bds_NoDeb0x803d :
STRUCT
	DTC: UDINT := 16#803D00;
	DFCid: UINT := 782;
	debounceMethod: USINT := NO_DEBOUNCE;
END_STRUCT
END_TYPE

// BODAS_RC18_12_40/Application/02 EasyConfig/DSM_easyConfig/Structure/DFC_bds_NoDeb0x803e
{attribute 'external_name' := 'cmp_rts_DFC_bds_NoDeb0x803e'}
TYPE DFC_bds_NoDeb0x803e :
STRUCT
	DTC: UDINT := 16#803E00;
	DFCid: UINT := 783;
	debounceMethod: USINT := NO_DEBOUNCE;
END_STRUCT
END_TYPE

// BODAS_RC18_12_40/Application/02 EasyConfig/DSM_easyConfig/Structure/DFC_bds_NoDeb0x803f
{attribute 'external_name' := 'cmp_rts_DFC_bds_NoDeb0x803f'}
TYPE DFC_bds_NoDeb0x803f : STRUCT
        DTC            : UDINT := 16#803F00;
        DFCid          : UINT  := 784;
        debounceMethod : USINT := NO_DEBOUNCE;
    END_STRUCT
END_TYPE

// BODAS_RC18_12_40/Application/02 EasyConfig/DSM_easyConfig/Structure/DFC_bds_NoDeb0x8040
{attribute 'external_name' := 'cmp_rts_DFC_bds_NoDeb0x8040'}
TYPE DFC_bds_NoDeb0x8040 : STRUCT
        DTC            : UDINT := 16#804000;
        DFCid          : UINT  := 785;
        debounceMethod : USINT := NO_DEBOUNCE;
    END_STRUCT
END_TYPE

// BODAS_RC18_12_40/Application/02 EasyConfig/DSM_easyConfig/Structure/DFC_bds_NoDeb0x8041
{attribute 'external_name' := 'cmp_rts_DFC_bds_NoDeb0x8041'}
TYPE DFC_bds_NoDeb0x8041 :
STRUCT
	DTC: UDINT := 16#804100;
	DFCid: UINT := 786;
	debounceMethod: USINT := NO_DEBOUNCE;
END_STRUCT
END_TYPE

// BODAS_RC18_12_40/Application/02 EasyConfig/DSM_easyConfig/Structure/DFC_bds_NoDeb0x8042
{attribute 'external_name' := 'cmp_rts_DFC_bds_NoDeb0x8042'}
TYPE DFC_bds_NoDeb0x8042 : STRUCT
        DTC            : UDINT := 16#804200;
        DFCid          : UINT  := 787;
        debounceMethod : USINT := NO_DEBOUNCE;
    END_STRUCT
END_TYPE

// BODAS_RC18_12_40/Application/02 EasyConfig/DSM_easyConfig/Structure/DFC_bds_NoDeb0x8043
{attribute 'external_name' := 'cmp_rts_DFC_bds_NoDeb0x8043'}
TYPE DFC_bds_NoDeb0x8043 :
STRUCT
	DTC: UDINT := 16#804300;
	DFCid: UINT := 788;
	debounceMethod: USINT := NO_DEBOUNCE;
END_STRUCT
END_TYPE

// BODAS_RC18_12_40/Application/02 EasyConfig/DSM_easyConfig/Structure/DFC_bds_NoDeb0x8044
{attribute 'external_name' := 'cmp_rts_DFC_bds_NoDeb0x8044'}
TYPE DFC_bds_NoDeb0x8044 : STRUCT
        DTC            : UDINT := 16#804400;
        DFCid          : UINT  := 789;
        debounceMethod : USINT := NO_DEBOUNCE;
    END_STRUCT
END_TYPE

// BODAS_RC18_12_40/Application/02 EasyConfig/DSM_easyConfig/Structure/DFC_bds_NoDeb0x8045
{attribute 'external_name' := 'cmp_rts_DFC_bds_NoDeb0x8045'}
TYPE DFC_bds_NoDeb0x8045 :
STRUCT
	DTC: UDINT := 16#804500;
	DFCid: UINT := 790;
	debounceMethod: USINT := NO_DEBOUNCE;
END_STRUCT
END_TYPE

// BODAS_RC18_12_40/Application/02 EasyConfig/DSM_easyConfig/Structure/DFC_bds_NoDeb0x8046
{attribute 'external_name' := 'cmp_rts_DFC_bds_NoDeb0x8046'}
TYPE DFC_bds_NoDeb0x8046 : STRUCT
        DTC            : UDINT := 16#804600;
        DFCid          : UINT  := 791;
        debounceMethod : USINT := NO_DEBOUNCE;
    END_STRUCT
END_TYPE

// BODAS_RC18_12_40/Application/02 EasyConfig/DSM_easyConfig/Structure/DFC_bds_NoDeb0x8047
{attribute 'external_name' := 'cmp_rts_DFC_bds_NoDeb0x8047'}
TYPE DFC_bds_NoDeb0x8047 : STRUCT
        DTC            : UDINT := 16#804700;
        DFCid          : UINT  := 792;
        debounceMethod : USINT := NO_DEBOUNCE;
    END_STRUCT
END_TYPE

// BODAS_RC18_12_40/Application/02 EasyConfig/DSM_easyConfig/Structure/DFC_bds_NoDeb0x8048
{attribute 'external_name' := 'cmp_rts_DFC_bds_NoDeb0x8048'}
TYPE DFC_bds_NoDeb0x8048 : STRUCT
        DTC            : UDINT := 16#804800;
        DFCid          : UINT  := 793;
        debounceMethod : USINT := NO_DEBOUNCE;
    END_STRUCT
END_TYPE

// BODAS_RC18_12_40/Application/02 EasyConfig/DSM_easyConfig/Structure/DFC_bds_NoDeb0x8049
{attribute 'external_name' := 'cmp_rts_DFC_bds_NoDeb0x8049'}
TYPE DFC_bds_NoDeb0x8049 : STRUCT
        DTC            : UDINT := 16#804900;
        DFCid          : UINT  := 794;
        debounceMethod : USINT := NO_DEBOUNCE;
    END_STRUCT
END_TYPE

// BODAS_RC18_12_40/Application/02 EasyConfig/DSM_easyConfig/Structure/DFC_bds_NoDeb0x804a
{attribute 'external_name' := 'cmp_rts_DFC_bds_NoDeb0x804a'}
TYPE DFC_bds_NoDeb0x804a : STRUCT
        DTC            : UDINT := 16#804A00;
        DFCid          : UINT  := 795;
        debounceMethod : USINT := NO_DEBOUNCE;
    END_STRUCT
END_TYPE

// BODAS_RC18_12_40/Application/02 EasyConfig/DSM_easyConfig/Structure/DFC_bds_NoDeb0x804b
{attribute 'external_name' := 'cmp_rts_DFC_bds_NoDeb0x804b'}
TYPE DFC_bds_NoDeb0x804b : STRUCT
        DTC            : UDINT := 16#804B00;
        DFCid          : UINT  := 796;
        debounceMethod : USINT := NO_DEBOUNCE;
    END_STRUCT
END_TYPE

// BODAS_RC18_12_40/Application/02 EasyConfig/DSM_easyConfig/Structure/DFC_bds_NoDeb0x804c
{attribute 'external_name' := 'cmp_rts_DFC_bds_NoDeb0x804c'}
TYPE DFC_bds_NoDeb0x804c : STRUCT
        DTC            : UDINT := 16#804C00;
        DFCid          : UINT  := 797;
        debounceMethod : USINT := NO_DEBOUNCE;
    END_STRUCT
END_TYPE

// BODAS_RC18_12_40/Application/02 EasyConfig/DSM_easyConfig/Structure/DFC_bds_NoDeb0x804d
{attribute 'external_name' := 'cmp_rts_DFC_bds_NoDeb0x804d'}
TYPE DFC_bds_NoDeb0x804d : STRUCT
        DTC            : UDINT := 16#804D00;
        DFCid          : UINT  := 798;
        debounceMethod : USINT := NO_DEBOUNCE;
    END_STRUCT
END_TYPE

// BODAS_RC18_12_40/Application/02 EasyConfig/DSM_easyConfig/Structure/DFC_bds_NoDeb0x804e
{attribute 'external_name' := 'cmp_rts_DFC_bds_NoDeb0x804e'}
TYPE DFC_bds_NoDeb0x804e : STRUCT
        DTC            : UDINT := 16#804E00;
        DFCid          : UINT  := 799;
        debounceMethod : USINT := NO_DEBOUNCE;
    END_STRUCT
END_TYPE

// BODAS_RC18_12_40/Application/02 EasyConfig/DSM_easyConfig/Structure/DFC_bds_NoDeb0x804f
{attribute 'external_name' := 'cmp_rts_DFC_bds_NoDeb0x804f'}
TYPE DFC_bds_NoDeb0x804f : STRUCT
        DTC            : UDINT := 16#804F00;
        DFCid          : UINT  := 800;
        debounceMethod : USINT := NO_DEBOUNCE;
    END_STRUCT
END_TYPE

// BODAS_RC18_12_40/Application/02 EasyConfig/DSM_easyConfig/Structure/DFC_bds_NoDeb0x8050
{attribute 'external_name' := 'cmp_rts_DFC_bds_NoDeb0x8050'}
TYPE DFC_bds_NoDeb0x8050 : STRUCT
        DTC            : UDINT := 16#805000;
        DFCid          : UINT  := 801;
        debounceMethod : USINT := NO_DEBOUNCE;
    END_STRUCT
END_TYPE

// BODAS_RC18_12_40/Application/02 EasyConfig/DSM_easyConfig/Structure/DFC_bds_NoDeb0x8051
{attribute 'external_name' := 'cmp_rts_DFC_bds_NoDeb0x8051'}
TYPE DFC_bds_NoDeb0x8051 :
STRUCT
	DTC: UDINT := 16#805100;
	DFCid: UINT := 802;
	debounceMethod: USINT := NO_DEBOUNCE;
END_STRUCT
END_TYPE

// BODAS_RC18_12_40/Application/02 EasyConfig/DSM_easyConfig/Structure/DFC_bds_NoDeb0x8052
{attribute 'external_name' := 'cmp_rts_DFC_bds_NoDeb0x8052'}
TYPE DFC_bds_NoDeb0x8052 : STRUCT
        DTC            : UDINT := 16#805200;
        DFCid          : UINT  := 803;
        debounceMethod : USINT := NO_DEBOUNCE;
    END_STRUCT
END_TYPE

// BODAS_RC18_12_40/Application/02 EasyConfig/DSM_easyConfig/Structure/DFC_bds_NoDeb0x8053
{attribute 'external_name' := 'cmp_rts_DFC_bds_NoDeb0x8053'}
TYPE DFC_bds_NoDeb0x8053 :
STRUCT
	DTC: UDINT := 16#805300;
	DFCid: UINT := 804;
	debounceMethod: USINT := NO_DEBOUNCE;
END_STRUCT
END_TYPE

// BODAS_RC18_12_40/Application/02 EasyConfig/DSM_easyConfig/Structure/DFC_bds_NoDeb0x8054
{attribute 'external_name' := 'cmp_rts_DFC_bds_NoDeb0x8054'}
TYPE DFC_bds_NoDeb0x8054 : STRUCT
        DTC            : UDINT := 16#805400;
        DFCid          : UINT  := 805;
        debounceMethod : USINT := NO_DEBOUNCE;
    END_STRUCT
END_TYPE

// BODAS_RC18_12_40/Application/02 EasyConfig/DSM_easyConfig/Structure/DFC_bds_NoDeb0x8055
{attribute 'external_name' := 'cmp_rts_DFC_bds_NoDeb0x8055'}
TYPE DFC_bds_NoDeb0x8055 : STRUCT
        DTC            : UDINT := 16#805500;
        DFCid          : UINT  := 806;
        debounceMethod : USINT := NO_DEBOUNCE;
    END_STRUCT
END_TYPE

// BODAS_RC18_12_40/Application/02 EasyConfig/DSM_easyConfig/Structure/DFC_bds_NoDeb0x8056
{attribute 'external_name' := 'cmp_rts_DFC_bds_NoDeb0x8056'}
TYPE DFC_bds_NoDeb0x8056 :
STRUCT
	DTC: UDINT := 16#805600;
	DFCid: UINT := 807;
	debounceMethod: USINT := NO_DEBOUNCE;
END_STRUCT
END_TYPE

// BODAS_RC18_12_40/Application/02 EasyConfig/DSM_easyConfig/Structure/DFC_bds_NoDeb0x8057
{attribute 'external_name' := 'cmp_rts_DFC_bds_NoDeb0x8057'}
TYPE DFC_bds_NoDeb0x8057 : STRUCT
        DTC            : UDINT := 16#805700;
        DFCid          : UINT  := 808;
        debounceMethod : USINT := NO_DEBOUNCE;
    END_STRUCT
END_TYPE

// BODAS_RC18_12_40/Application/02 EasyConfig/DSM_easyConfig/Structure/DFC_bds_NoDeb0x8058
{attribute 'external_name' := 'cmp_rts_DFC_bds_NoDeb0x8058'}
TYPE DFC_bds_NoDeb0x8058 : STRUCT
        DTC            : UDINT := 16#805800;
        DFCid          : UINT  := 809;
        debounceMethod : USINT := NO_DEBOUNCE;
    END_STRUCT
END_TYPE

// BODAS_RC18_12_40/Application/02 EasyConfig/DSM_easyConfig/Structure/DFC_bds_NoDeb0x8059
{attribute 'external_name' := 'cmp_rts_DFC_bds_NoDeb0x8059'}
TYPE DFC_bds_NoDeb0x8059 :
STRUCT
	DTC: UDINT := 16#805900;
	DFCid: UINT := 810;
	debounceMethod: USINT := NO_DEBOUNCE;
END_STRUCT
END_TYPE

// BODAS_RC18_12_40/Application/02 EasyConfig/DSM_easyConfig/Structure/DFC_bds_NoDeb0x805a
{attribute 'external_name' := 'cmp_rts_DFC_bds_NoDeb0x805a'}
TYPE DFC_bds_NoDeb0x805a :
STRUCT
	DTC: UDINT := 16#805A00;
	DFCid: UINT := 811;
	debounceMethod: USINT := NO_DEBOUNCE;
END_STRUCT
END_TYPE

// BODAS_RC18_12_40/Application/02 EasyConfig/DSM_easyConfig/Structure/DFC_bds_NoDeb0x805b
{attribute 'external_name' := 'cmp_rts_DFC_bds_NoDeb0x805b'}
TYPE DFC_bds_NoDeb0x805b : STRUCT
        DTC            : UDINT := 16#805B00;
        DFCid          : UINT  := 812;
        debounceMethod : USINT := NO_DEBOUNCE;
    END_STRUCT
END_TYPE

// BODAS_RC18_12_40/Application/02 EasyConfig/DSM_easyConfig/Structure/DFC_bds_NoDeb0x805c
{attribute 'external_name' := 'cmp_rts_DFC_bds_NoDeb0x805c'}
TYPE DFC_bds_NoDeb0x805c : STRUCT
        DTC            : UDINT := 16#805C00;
        DFCid          : UINT  := 813;
        debounceMethod : USINT := NO_DEBOUNCE;
    END_STRUCT
END_TYPE

// BODAS_RC18_12_40/Application/02 EasyConfig/DSM_easyConfig/Structure/DFC_bds_NoDeb0x805d
{attribute 'external_name' := 'cmp_rts_DFC_bds_NoDeb0x805d'}
TYPE DFC_bds_NoDeb0x805d : STRUCT
        DTC            : UDINT := 16#805D00;
        DFCid          : UINT  := 814;
        debounceMethod : USINT := NO_DEBOUNCE;
    END_STRUCT
END_TYPE

// BODAS_RC18_12_40/Application/02 EasyConfig/DSM_easyConfig/Structure/DFC_bds_NoDeb0x805e
{attribute 'external_name' := 'cmp_rts_DFC_bds_NoDeb0x805e'}
TYPE DFC_bds_NoDeb0x805e : STRUCT
        DTC            : UDINT := 16#805E00;
        DFCid          : UINT  := 815;
        debounceMethod : USINT := NO_DEBOUNCE;
    END_STRUCT
END_TYPE

// BODAS_RC18_12_40/Application/02 EasyConfig/DSM_easyConfig/Structure/DFC_bds_NoDeb0x805f
{attribute 'external_name' := 'cmp_rts_DFC_bds_NoDeb0x805f'}
TYPE DFC_bds_NoDeb0x805f : STRUCT
        DTC            : UDINT := 16#805F00;
        DFCid          : UINT  := 816;
        debounceMethod : USINT := NO_DEBOUNCE;
    END_STRUCT
END_TYPE

// BODAS_RC18_12_40/Application/02 EasyConfig/DSM_easyConfig/Structure/DFC_bds_NoDeb0x8060
{attribute 'external_name' := 'cmp_rts_DFC_bds_NoDeb0x8060'}
TYPE DFC_bds_NoDeb0x8060 :
STRUCT
	DTC: UDINT := 16#806000;
	DFCid: UINT := 817;
	debounceMethod: USINT := NO_DEBOUNCE;
END_STRUCT
END_TYPE

// BODAS_RC18_12_40/Application/02 EasyConfig/DSM_easyConfig/Structure/DFC_bds_NoDeb0x8061
{attribute 'external_name' := 'cmp_rts_DFC_bds_NoDeb0x8061'}
TYPE DFC_bds_NoDeb0x8061 : STRUCT
        DTC            : UDINT := 16#806100;
        DFCid          : UINT  := 818;
        debounceMethod : USINT := NO_DEBOUNCE;
    END_STRUCT
END_TYPE

// BODAS_RC18_12_40/Application/02 EasyConfig/DSM_easyConfig/Structure/DFC_bds_NoDeb0x8062
{attribute 'external_name' := 'cmp_rts_DFC_bds_NoDeb0x8062'}
TYPE DFC_bds_NoDeb0x8062 : STRUCT
        DTC            : UDINT := 16#806200;
        DFCid          : UINT  := 819;
        debounceMethod : USINT := NO_DEBOUNCE;
    END_STRUCT
END_TYPE

// BODAS_RC18_12_40/Application/02 EasyConfig/DSM_easyConfig/Structure/DFC_bds_NoDeb0x8063
{attribute 'external_name' := 'cmp_rts_DFC_bds_NoDeb0x8063'}
TYPE DFC_bds_NoDeb0x8063 : STRUCT
        DTC            : UDINT := 16#806300;
        DFCid          : UINT  := 106;
        debounceMethod : USINT := TIME_UP_DOWN;
    END_STRUCT
END_TYPE

// BODAS_RC18_12_40/Application/02 EasyConfig/DSM_easyConfig/Structure/DFC_bds_NoDeb0x8064
{attribute 'external_name' := 'cmp_rts_DFC_bds_NoDeb0x8064'}
TYPE DFC_bds_NoDeb0x8064 :
STRUCT
	DTC: UDINT := 16#806400;
	DFCid: UINT := 107;
	debounceMethod: USINT := TIME_UP_DOWN;
END_STRUCT
END_TYPE

// BODAS_RC18_12_40/Application/02 EasyConfig/DSM_easyConfig/Structure/DFC_bds_NoDeb0x8065
{attribute 'external_name' := 'cmp_rts_DFC_bds_NoDeb0x8065'}
TYPE DFC_bds_NoDeb0x8065 : STRUCT
        DTC            : UDINT := 16#806500;
        DFCid          : UINT  := 108;
        debounceMethod : USINT := TIME_UP_DOWN;
    END_STRUCT
END_TYPE

// BODAS_RC18_12_40/Application/02 EasyConfig/DSM_easyConfig/Structure/DFC_bds_NoDeb0x8066
{attribute 'external_name' := 'cmp_rts_DFC_bds_NoDeb0x8066'}
TYPE DFC_bds_NoDeb0x8066 : STRUCT
        DTC            : UDINT := 16#806600;
        DFCid          : UINT  := 109;
        debounceMethod : USINT := TIME_UP_DOWN;
    END_STRUCT
END_TYPE

// BODAS_RC18_12_40/Application/02 EasyConfig/DSM_easyConfig/Structure/DFC_bds_NoDeb0x8067
{attribute 'external_name' := 'cmp_rts_DFC_bds_NoDeb0x8067'}
TYPE DFC_bds_NoDeb0x8067 : STRUCT
        DTC            : UDINT := 16#806700;
        DFCid          : UINT  := 110;
        debounceMethod : USINT := TIME_UP_DOWN;
    END_STRUCT
END_TYPE

// BODAS_RC18_12_40/Application/02 EasyConfig/DSM_easyConfig/Structure/DFC_bds_NoDeb0x8068
{attribute 'external_name' := 'cmp_rts_DFC_bds_NoDeb0x8068'}
TYPE DFC_bds_NoDeb0x8068 : STRUCT
        DTC            : UDINT := 16#806800;
        DFCid          : UINT  := 111;
        debounceMethod : USINT := TIME_UP_DOWN;
    END_STRUCT
END_TYPE

// BODAS_RC18_12_40/Application/02 EasyConfig/DSM_easyConfig/Structure/DFC_bds_NoDeb0x8069
{attribute 'external_name' := 'cmp_rts_DFC_bds_NoDeb0x8069'}
TYPE DFC_bds_NoDeb0x8069 :
STRUCT
	DTC: UDINT := 16#806900;
	DFCid: UINT := 112;
	debounceMethod: USINT := TIME_UP_DOWN;
END_STRUCT
END_TYPE

// BODAS_RC18_12_40/Application/02 EasyConfig/DSM_easyConfig/Structure/DFC_bds_NoDeb0x806a
{attribute 'external_name' := 'cmp_rts_DFC_bds_NoDeb0x806a'}
TYPE DFC_bds_NoDeb0x806a : STRUCT
        DTC            : UDINT := 16#806A00;
        DFCid          : UINT  := 113;
        debounceMethod : USINT := TIME_UP_DOWN;
    END_STRUCT
END_TYPE

// BODAS_RC18_12_40/Application/02 EasyConfig/DSM_easyConfig/Structure/DFC_bds_NoDeb0x806b
{attribute 'external_name' := 'cmp_rts_DFC_bds_NoDeb0x806b'}
TYPE DFC_bds_NoDeb0x806b : STRUCT
        DTC            : UDINT := 16#806B00;
        DFCid          : UINT  := 114;
        debounceMethod : USINT := TIME_UP_DOWN;
    END_STRUCT
END_TYPE

// BODAS_RC18_12_40/Application/02 EasyConfig/DSM_easyConfig/Structure/DFC_bds_NoDeb0x806c
{attribute 'external_name' := 'cmp_rts_DFC_bds_NoDeb0x806c'}
TYPE DFC_bds_NoDeb0x806c : STRUCT
        DTC            : UDINT := 16#806C00;
        DFCid          : UINT  := 115;
        debounceMethod : USINT := TIME_UP_DOWN;
    END_STRUCT
END_TYPE

// BODAS_RC18_12_40/Application/02 EasyConfig/DSM_easyConfig/Structure/DFC_bds_NoDeb0x806d
{attribute 'external_name' := 'cmp_rts_DFC_bds_NoDeb0x806d'}
TYPE DFC_bds_NoDeb0x806d : STRUCT
        DTC            : UDINT := 16#806D00;
        DFCid          : UINT  := 116;
        debounceMethod : USINT := TIME_UP_DOWN;
    END_STRUCT
END_TYPE

// BODAS_RC18_12_40/Application/02 EasyConfig/DSM_easyConfig/Structure/DFC_bds_NoDeb0x806e
{attribute 'external_name' := 'cmp_rts_DFC_bds_NoDeb0x806e'}
TYPE DFC_bds_NoDeb0x806e : STRUCT
        DTC            : UDINT := 16#806E00;
        DFCid          : UINT  := 117;
        debounceMethod : USINT := TIME_UP_DOWN;
    END_STRUCT
END_TYPE

// BODAS_RC18_12_40/Application/02 EasyConfig/DSM_easyConfig/Structure/DFC_bds_NoDeb0x806f
{attribute 'external_name' := 'cmp_rts_DFC_bds_NoDeb0x806f'}
TYPE DFC_bds_NoDeb0x806f :
STRUCT
	DTC: UDINT := 16#806F00;
	DFCid: UINT := 118;
	debounceMethod: USINT := TIME_UP_DOWN;
END_STRUCT
END_TYPE

// BODAS_RC18_12_40/Application/02 EasyConfig/DSM_easyConfig/Structure/DFC_bds_NoDeb0x8070
{attribute 'external_name' := 'cmp_rts_DFC_bds_NoDeb0x8070'}
TYPE DFC_bds_NoDeb0x8070 : STRUCT
        DTC            : UDINT := 16#807000;
        DFCid          : UINT  := 119;
        debounceMethod : USINT := TIME_UP_DOWN;
    END_STRUCT
END_TYPE

// BODAS_RC18_12_40/Application/02 EasyConfig/DSM_easyConfig/Structure/DFC_bds_NoDeb0x8071
{attribute 'external_name' := 'cmp_rts_DFC_bds_NoDeb0x8071'}
TYPE DFC_bds_NoDeb0x8071 : STRUCT
        DTC            : UDINT := 16#807100;
        DFCid          : UINT  := 120;
        debounceMethod : USINT := TIME_UP_DOWN;
    END_STRUCT
END_TYPE

// BODAS_RC18_12_40/Application/02 EasyConfig/DSM_easyConfig/Structure/DFC_bds_NoDeb0x8072
{attribute 'external_name' := 'cmp_rts_DFC_bds_NoDeb0x8072'}
TYPE DFC_bds_NoDeb0x8072 : STRUCT
        DTC            : UDINT := 16#807200;
        DFCid          : UINT  := 121;
        debounceMethod : USINT := TIME_UP_DOWN;
    END_STRUCT
END_TYPE

// BODAS_RC18_12_40/Application/02 EasyConfig/DSM_easyConfig/Structure/DFC_bds_NoDeb0x8073
{attribute 'external_name' := 'cmp_rts_DFC_bds_NoDeb0x8073'}
TYPE DFC_bds_NoDeb0x8073 :
STRUCT
	DTC: UDINT := 16#807300;
	DFCid: UINT := 122;
	debounceMethod: USINT := TIME_UP_DOWN;
END_STRUCT
END_TYPE

// BODAS_RC18_12_40/Application/02 EasyConfig/DSM_easyConfig/Structure/DFC_bds_NoDeb0x8074
{attribute 'external_name' := 'cmp_rts_DFC_bds_NoDeb0x8074'}
TYPE DFC_bds_NoDeb0x8074 : STRUCT
        DTC            : UDINT := 16#807400;
        DFCid          : UINT  := 123;
        debounceMethod : USINT := TIME_UP_DOWN;
    END_STRUCT
END_TYPE

// BODAS_RC18_12_40/Application/02 EasyConfig/DSM_easyConfig/Structure/DFC_bds_NoDeb0x8075
{attribute 'external_name' := 'cmp_rts_DFC_bds_NoDeb0x8075'}
TYPE DFC_bds_NoDeb0x8075 : STRUCT
        DTC            : UDINT := 16#807500;
        DFCid          : UINT  := 124;
        debounceMethod : USINT := TIME_UP_DOWN;
    END_STRUCT
END_TYPE

// BODAS_RC18_12_40/Application/02 EasyConfig/DSM_easyConfig/Structure/DFC_bds_NoDeb0x8076
{attribute 'external_name' := 'cmp_rts_DFC_bds_NoDeb0x8076'}
TYPE DFC_bds_NoDeb0x8076 : STRUCT
        DTC            : UDINT := 16#807600;
        DFCid          : UINT  := 125;
        debounceMethod : USINT := TIME_UP_DOWN;
    END_STRUCT
END_TYPE

// BODAS_RC18_12_40/Application/02 EasyConfig/DSM_easyConfig/Structure/DFC_bds_NoDeb0x8077
{attribute 'external_name' := 'cmp_rts_DFC_bds_NoDeb0x8077'}
TYPE DFC_bds_NoDeb0x8077 : STRUCT
        DTC            : UDINT := 16#807700;
        DFCid          : UINT  := 126;
        debounceMethod : USINT := TIME_UP_DOWN;
    END_STRUCT
END_TYPE

// BODAS_RC18_12_40/Application/02 EasyConfig/DSM_easyConfig/Structure/DFC_bds_NoDeb0x8078
{attribute 'external_name' := 'cmp_rts_DFC_bds_NoDeb0x8078'}
TYPE DFC_bds_NoDeb0x8078 : STRUCT
        DTC            : UDINT := 16#807800;
        DFCid          : UINT  := 127;
        debounceMethod : USINT := TIME_UP_DOWN;
    END_STRUCT
END_TYPE

// BODAS_RC18_12_40/Application/02 EasyConfig/DSM_easyConfig/Structure/DFC_bds_NoDeb0x8079
{attribute 'external_name' := 'cmp_rts_DFC_bds_NoDeb0x8079'}
TYPE DFC_bds_NoDeb0x8079 : STRUCT
        DTC            : UDINT := 16#807900;
        DFCid          : UINT  := 128;
        debounceMethod : USINT := TIME_UP_DOWN;
    END_STRUCT
END_TYPE

// BODAS_RC18_12_40/Application/02 EasyConfig/DSM_easyConfig/Structure/DFC_bds_NoDeb0x807a
{attribute 'external_name' := 'cmp_rts_DFC_bds_NoDeb0x807a'}
TYPE DFC_bds_NoDeb0x807a : STRUCT
        DTC            : UDINT := 16#807A00;
        DFCid          : UINT  := 129;
        debounceMethod : USINT := TIME_UP_DOWN;
    END_STRUCT
END_TYPE

// BODAS_RC18_12_40/Application/02 EasyConfig/DSM_easyConfig/Structure/DFC_bds_NoDeb0x807b
{attribute 'external_name' := 'cmp_rts_DFC_bds_NoDeb0x807b'}
TYPE DFC_bds_NoDeb0x807b : STRUCT
        DTC            : UDINT := 16#807B00;
        DFCid          : UINT  := 130;
        debounceMethod : USINT := TIME_UP_DOWN;
    END_STRUCT
END_TYPE

// BODAS_RC18_12_40/Application/02 EasyConfig/DSM_easyConfig/Structure/DFC_bds_NoDeb0x807c
{attribute 'external_name' := 'cmp_rts_DFC_bds_NoDeb0x807c'}
TYPE DFC_bds_NoDeb0x807c : STRUCT
        DTC            : UDINT := 16#807C00;
        DFCid          : UINT  := 131;
        debounceMethod : USINT := TIME_UP_DOWN;
    END_STRUCT
END_TYPE

// BODAS_RC18_12_40/Application/02 EasyConfig/DSM_easyConfig/Structure/DFC_bds_NoDeb0x807d
{attribute 'external_name' := 'cmp_rts_DFC_bds_NoDeb0x807d'}
TYPE DFC_bds_NoDeb0x807d : STRUCT
        DTC            : UDINT := 16#807D00;
        DFCid          : UINT  := 132;
        debounceMethod : USINT := TIME_UP_DOWN;
    END_STRUCT
END_TYPE

// BODAS_RC18_12_40/Application/02 EasyConfig/DSM_easyConfig/Structure/DFC_bds_NoDeb0x807e
{attribute 'external_name' := 'cmp_rts_DFC_bds_NoDeb0x807e'}
TYPE DFC_bds_NoDeb0x807e : STRUCT
        DTC            : UDINT := 16#807E00;
        DFCid          : UINT  := 133;
        debounceMethod : USINT := TIME_UP_DOWN;
    END_STRUCT
END_TYPE

// BODAS_RC18_12_40/Application/02 EasyConfig/DSM_easyConfig/Structure/DFC_bds_NoDeb0x807f
{attribute 'external_name' := 'cmp_rts_DFC_bds_NoDeb0x807f'}
TYPE DFC_bds_NoDeb0x807f : STRUCT
        DTC            : UDINT := 16#807F00;
        DFCid          : UINT  := 134;
        debounceMethod : USINT := TIME_UP_DOWN;
    END_STRUCT
END_TYPE

// BODAS_RC18_12_40/Application/02 EasyConfig/DSM_easyConfig/Structure/DFC_bds_NoDeb0x8080
{attribute 'external_name' := 'cmp_rts_DFC_bds_NoDeb0x8080'}
TYPE DFC_bds_NoDeb0x8080 : STRUCT
        DTC            : UDINT := 16#808000;
        DFCid          : UINT  := 135;
        debounceMethod : USINT := TIME_UP_DOWN;
    END_STRUCT
END_TYPE

// BODAS_RC18_12_40/Application/02 EasyConfig/DSM_easyConfig/Structure/DFC_bds_NoDeb0x8081
{attribute 'external_name' := 'cmp_rts_DFC_bds_NoDeb0x8081'}
TYPE DFC_bds_NoDeb0x8081 : STRUCT
        DTC            : UDINT := 16#808100;
        DFCid          : UINT  := 136;
        debounceMethod : USINT := TIME_UP_DOWN;
    END_STRUCT
END_TYPE

// BODAS_RC18_12_40/Application/02 EasyConfig/DSM_easyConfig/Structure/DFC_bds_NoDeb0x8082
{attribute 'external_name' := 'cmp_rts_DFC_bds_NoDeb0x8082'}
TYPE DFC_bds_NoDeb0x8082 : STRUCT
        DTC            : UDINT := 16#808200;
        DFCid          : UINT  := 137;
        debounceMethod : USINT := TIME_UP_DOWN;
    END_STRUCT
END_TYPE

// BODAS_RC18_12_40/Application/02 EasyConfig/DSM_easyConfig/Structure/DFC_bds_NoDeb0x8083
{attribute 'external_name' := 'cmp_rts_DFC_bds_NoDeb0x8083'}
TYPE DFC_bds_NoDeb0x8083 : STRUCT
        DTC            : UDINT := 16#808300;
        DFCid          : UINT  := 138;
        debounceMethod : USINT := TIME_UP_DOWN;
    END_STRUCT
END_TYPE

// BODAS_RC18_12_40/Application/02 EasyConfig/DSM_easyConfig/Structure/DFC_bds_NoDeb0x8084
{attribute 'external_name' := 'cmp_rts_DFC_bds_NoDeb0x8084'}
TYPE DFC_bds_NoDeb0x8084 : STRUCT
        DTC            : UDINT := 16#808400;
        DFCid          : UINT  := 139;
        debounceMethod : USINT := TIME_UP_DOWN;
    END_STRUCT
END_TYPE

// BODAS_RC18_12_40/Application/02 EasyConfig/DSM_easyConfig/Structure/DFC_bds_NoDeb0x8085
{attribute 'external_name' := 'cmp_rts_DFC_bds_NoDeb0x8085'}
TYPE DFC_bds_NoDeb0x8085 : STRUCT
        DTC            : UDINT := 16#808500;
        DFCid          : UINT  := 140;
        debounceMethod : USINT := TIME_UP_DOWN;
    END_STRUCT
END_TYPE

// BODAS_RC18_12_40/Application/02 EasyConfig/DSM_easyConfig/Structure/DFC_bds_NoDeb0x8086
{attribute 'external_name' := 'cmp_rts_DFC_bds_NoDeb0x8086'}
TYPE DFC_bds_NoDeb0x8086 : STRUCT
        DTC            : UDINT := 16#808600;
        DFCid          : UINT  := 141;
        debounceMethod : USINT := TIME_UP_DOWN;
    END_STRUCT
END_TYPE

// BODAS_RC18_12_40/Application/02 EasyConfig/DSM_easyConfig/Structure/DFC_bds_NoDeb0x8087
{attribute 'external_name' := 'cmp_rts_DFC_bds_NoDeb0x8087'}
TYPE DFC_bds_NoDeb0x8087 : STRUCT
        DTC            : UDINT := 16#808700;
        DFCid          : UINT  := 142;
        debounceMethod : USINT := TIME_UP_DOWN;
    END_STRUCT
END_TYPE

// BODAS_RC18_12_40/Application/02 EasyConfig/DSM_easyConfig/Structure/DFC_bds_NoDeb0x8088
{attribute 'external_name' := 'cmp_rts_DFC_bds_NoDeb0x8088'}
TYPE DFC_bds_NoDeb0x8088 : STRUCT
        DTC            : UDINT := 16#808800;
        DFCid          : UINT  := 143;
        debounceMethod : USINT := TIME_UP_DOWN;
    END_STRUCT
END_TYPE

// BODAS_RC18_12_40/Application/02 EasyConfig/DSM_easyConfig/Structure/DFC_bds_NoDeb0x8089
{attribute 'external_name' := 'cmp_rts_DFC_bds_NoDeb0x8089'}
TYPE DFC_bds_NoDeb0x8089 : STRUCT
        DTC            : UDINT := 16#808900;
        DFCid          : UINT  := 144;
        debounceMethod : USINT := TIME_UP_DOWN;
    END_STRUCT
END_TYPE

// BODAS_RC18_12_40/Application/02 EasyConfig/DSM_easyConfig/Structure/DFC_bds_NoDeb0x808a
{attribute 'external_name' := 'cmp_rts_DFC_bds_NoDeb0x808a'}
TYPE DFC_bds_NoDeb0x808a : STRUCT
        DTC            : UDINT := 16#808A00;
        DFCid          : UINT  := 145;
        debounceMethod : USINT := TIME_UP_DOWN;
    END_STRUCT
END_TYPE

// BODAS_RC18_12_40/Application/02 EasyConfig/DSM_easyConfig/Structure/DFC_bds_NoDeb0x808b
{attribute 'external_name' := 'cmp_rts_DFC_bds_NoDeb0x808b'}
TYPE DFC_bds_NoDeb0x808b : STRUCT
        DTC            : UDINT := 16#808B00;
        DFCid          : UINT  := 146;
        debounceMethod : USINT := TIME_UP_DOWN;
    END_STRUCT
END_TYPE

// BODAS_RC18_12_40/Application/02 EasyConfig/DSM_easyConfig/Structure/DFC_bds_NoDeb0x808c
{attribute 'external_name' := 'cmp_rts_DFC_bds_NoDeb0x808c'}
TYPE DFC_bds_NoDeb0x808c : STRUCT
        DTC            : UDINT := 16#808C00;
        DFCid          : UINT  := 147;
        debounceMethod : USINT := TIME_UP_DOWN;
    END_STRUCT
END_TYPE

// BODAS_RC18_12_40/Application/02 EasyConfig/DSM_easyConfig/Structure/DFC_bds_NoDeb0x808d
{attribute 'external_name' := 'cmp_rts_DFC_bds_NoDeb0x808d'}
TYPE DFC_bds_NoDeb0x808d : STRUCT
        DTC            : UDINT := 16#808D00;
        DFCid          : UINT  := 148;
        debounceMethod : USINT := TIME_UP_DOWN;
    END_STRUCT
END_TYPE

// BODAS_RC18_12_40/Application/02 EasyConfig/DSM_easyConfig/Structure/DFC_bds_NoDeb0x808e
{attribute 'external_name' := 'cmp_rts_DFC_bds_NoDeb0x808e'}
TYPE DFC_bds_NoDeb0x808e : STRUCT
        DTC            : UDINT := 16#808E00;
        DFCid          : UINT  := 149;
        debounceMethod : USINT := TIME_UP_DOWN;
    END_STRUCT
END_TYPE

// BODAS_RC18_12_40/Application/02 EasyConfig/DSM_easyConfig/Structure/DFC_bds_NoDeb0x808f
{attribute 'external_name' := 'cmp_rts_DFC_bds_NoDeb0x808f'}
TYPE DFC_bds_NoDeb0x808f : STRUCT
        DTC            : UDINT := 16#808F00;
        DFCid          : UINT  := 150;
        debounceMethod : USINT := TIME_UP_DOWN;
    END_STRUCT
END_TYPE

// BODAS_RC18_12_40/Application/02 EasyConfig/DSM_easyConfig/Structure/DFC_bds_NoDeb0x8090
{attribute 'external_name' := 'cmp_rts_DFC_bds_NoDeb0x8090'}
TYPE DFC_bds_NoDeb0x8090 : STRUCT
        DTC            : UDINT := 16#809000;
        DFCid          : UINT  := 151;
        debounceMethod : USINT := TIME_UP_DOWN;
    END_STRUCT
END_TYPE

// BODAS_RC18_12_40/Application/02 EasyConfig/DSM_easyConfig/Structure/DFC_bds_NoDeb0x8091
{attribute 'external_name' := 'cmp_rts_DFC_bds_NoDeb0x8091'}
TYPE DFC_bds_NoDeb0x8091 : STRUCT
        DTC            : UDINT := 16#809100;
        DFCid          : UINT  := 152;
        debounceMethod : USINT := TIME_UP_DOWN;
    END_STRUCT
END_TYPE

// BODAS_RC18_12_40/Application/02 EasyConfig/DSM_easyConfig/Structure/DFC_bds_NoDeb0x8092
{attribute 'external_name' := 'cmp_rts_DFC_bds_NoDeb0x8092'}
TYPE DFC_bds_NoDeb0x8092 : STRUCT
        DTC            : UDINT := 16#809200;
        DFCid          : UINT  := 153;
        debounceMethod : USINT := TIME_UP_DOWN;
    END_STRUCT
END_TYPE

// BODAS_RC18_12_40/Application/02 EasyConfig/DSM_easyConfig/Structure/DFC_bds_NoDeb0x8093
{attribute 'external_name' := 'cmp_rts_DFC_bds_NoDeb0x8093'}
TYPE DFC_bds_NoDeb0x8093 : STRUCT
        DTC            : UDINT := 16#809300;
        DFCid          : UINT  := 154;
        debounceMethod : USINT := TIME_UP_DOWN;
    END_STRUCT
END_TYPE

// BODAS_RC18_12_40/Application/02 EasyConfig/DSM_easyConfig/Structure/DFC_bds_NoDeb0x8094
{attribute 'external_name' := 'cmp_rts_DFC_bds_NoDeb0x8094'}
TYPE DFC_bds_NoDeb0x8094 : STRUCT
        DTC            : UDINT := 16#809400;
        DFCid          : UINT  := 155;
        debounceMethod : USINT := TIME_UP_DOWN;
    END_STRUCT
END_TYPE

// BODAS_RC18_12_40/Application/02 EasyConfig/DSM_easyConfig/Structure/DFC_bds_NoDeb0x8095
{attribute 'external_name' := 'cmp_rts_DFC_bds_NoDeb0x8095'}
TYPE DFC_bds_NoDeb0x8095 : STRUCT
        DTC            : UDINT := 16#809500;
        DFCid          : UINT  := 156;
        debounceMethod : USINT := TIME_UP_DOWN;
    END_STRUCT
END_TYPE

// BODAS_RC18_12_40/Application/02 EasyConfig/DSM_easyConfig/Structure/DFC_bds_NoDeb0x8096
{attribute 'external_name' := 'cmp_rts_DFC_bds_NoDeb0x8096'}
TYPE DFC_bds_NoDeb0x8096 : STRUCT
        DTC            : UDINT := 16#809600;
        DFCid          : UINT  := 157;
        debounceMethod : USINT := TIME_UP_DOWN;
    END_STRUCT
END_TYPE

// BODAS_RC18_12_40/Application/02 EasyConfig/DSM_easyConfig/Structure/DFC_bds_NoDeb0x8097
{attribute 'external_name' := 'cmp_rts_DFC_bds_NoDeb0x8097'}
TYPE DFC_bds_NoDeb0x8097 : STRUCT
        DTC            : UDINT := 16#809700;
        DFCid          : UINT  := 158;
        debounceMethod : USINT := TIME_UP_DOWN;
    END_STRUCT
END_TYPE

// BODAS_RC18_12_40/Application/02 EasyConfig/DSM_easyConfig/Structure/DFC_bds_NoDeb0x8098
{attribute 'external_name' := 'cmp_rts_DFC_bds_NoDeb0x8098'}
TYPE DFC_bds_NoDeb0x8098 : STRUCT
        DTC            : UDINT := 16#809800;
        DFCid          : UINT  := 159;
        debounceMethod : USINT := TIME_UP_DOWN;
    END_STRUCT
END_TYPE

// BODAS_RC18_12_40/Application/02 EasyConfig/DSM_easyConfig/Structure/DFC_bds_NoDeb0x8099
{attribute 'external_name' := 'cmp_rts_DFC_bds_NoDeb0x8099'}
TYPE DFC_bds_NoDeb0x8099 : STRUCT
        DTC            : UDINT := 16#809900;
        DFCid          : UINT  := 160;
        debounceMethod : USINT := TIME_UP_DOWN;
    END_STRUCT
END_TYPE

// BODAS_RC18_12_40/Application/02 EasyConfig/DSM_easyConfig/Structure/DFC_bds_NoDeb0x809a
{attribute 'external_name' := 'cmp_rts_DFC_bds_NoDeb0x809a'}
TYPE DFC_bds_NoDeb0x809a : STRUCT
        DTC            : UDINT := 16#809A00;
        DFCid          : UINT  := 161;
        debounceMethod : USINT := TIME_UP_DOWN;
    END_STRUCT
END_TYPE

// BODAS_RC18_12_40/Application/02 EasyConfig/DSM_easyConfig/Structure/DFC_bds_NoDeb0x809b
{attribute 'external_name' := 'cmp_rts_DFC_bds_NoDeb0x809b'}
TYPE DFC_bds_NoDeb0x809b : STRUCT
        DTC            : UDINT := 16#809B00;
        DFCid          : UINT  := 162;
        debounceMethod : USINT := TIME_UP_DOWN;
    END_STRUCT
END_TYPE

// BODAS_RC18_12_40/Application/02 EasyConfig/DSM_easyConfig/Structure/DFC_bds_NoDeb0x809c
{attribute 'external_name' := 'cmp_rts_DFC_bds_NoDeb0x809c'}
TYPE DFC_bds_NoDeb0x809c : STRUCT
        DTC            : UDINT := 16#809C00;
        DFCid          : UINT  := 163;
        debounceMethod : USINT := TIME_UP_DOWN;
    END_STRUCT
END_TYPE

// BODAS_RC18_12_40/Application/02 EasyConfig/DSM_easyConfig/Structure/DFC_bds_NoDeb0x809d
{attribute 'external_name' := 'cmp_rts_DFC_bds_NoDeb0x809d'}
TYPE DFC_bds_NoDeb0x809d : STRUCT
        DTC            : UDINT := 16#809D00;
        DFCid          : UINT  := 164;
        debounceMethod : USINT := TIME_UP_DOWN;
    END_STRUCT
END_TYPE

// BODAS_RC18_12_40/Application/02 EasyConfig/DSM_easyConfig/Structure/DFC_bds_NoDeb0x809e
{attribute 'external_name' := 'cmp_rts_DFC_bds_NoDeb0x809e'}
TYPE DFC_bds_NoDeb0x809e : STRUCT
        DTC            : UDINT := 16#809E00;
        DFCid          : UINT  := 165;
        debounceMethod : USINT := TIME_UP_DOWN;
    END_STRUCT
END_TYPE

// BODAS_RC18_12_40/Application/02 EasyConfig/DSM_easyConfig/Structure/DFC_bds_NoDeb0x809f
{attribute 'external_name' := 'cmp_rts_DFC_bds_NoDeb0x809f'}
TYPE DFC_bds_NoDeb0x809f : STRUCT
        DTC            : UDINT := 16#809F00;
        DFCid          : UINT  := 166;
        debounceMethod : USINT := TIME_UP_DOWN;
    END_STRUCT
END_TYPE

// BODAS_RC18_12_40/Application/02 EasyConfig/DSM_easyConfig/Structure/DFC_bds_NoDeb0x80a0
{attribute 'external_name' := 'cmp_rts_DFC_bds_NoDeb0x80a0'}
TYPE DFC_bds_NoDeb0x80a0 : STRUCT
        DTC            : UDINT := 16#80A000;
        DFCid          : UINT  := 167;
        debounceMethod : USINT := TIME_UP_DOWN;
    END_STRUCT
END_TYPE

// BODAS_RC18_12_40/Application/02 EasyConfig/DSM_easyConfig/Structure/DFC_bds_NoDeb0x80a1
{attribute 'external_name' := 'cmp_rts_DFC_bds_NoDeb0x80a1'}
TYPE DFC_bds_NoDeb0x80a1 : STRUCT
        DTC            : UDINT := 16#80A100;
        DFCid          : UINT  := 168;
        debounceMethod : USINT := TIME_UP_DOWN;
    END_STRUCT
END_TYPE

// BODAS_RC18_12_40/Application/02 EasyConfig/DSM_easyConfig/Structure/DFC_bds_NoDeb0x80a2
{attribute 'external_name' := 'cmp_rts_DFC_bds_NoDeb0x80a2'}
TYPE DFC_bds_NoDeb0x80a2 : STRUCT
        DTC            : UDINT := 16#80A200;
        DFCid          : UINT  := 169;
        debounceMethod : USINT := TIME_UP_DOWN;
    END_STRUCT
END_TYPE

// BODAS_RC18_12_40/Application/02 EasyConfig/DSM_easyConfig/Structure/DFC_bds_NoDeb0x80a3
{attribute 'external_name' := 'cmp_rts_DFC_bds_NoDeb0x80a3'}
TYPE DFC_bds_NoDeb0x80a3 : STRUCT
        DTC            : UDINT := 16#80A300;
        DFCid          : UINT  := 170;
        debounceMethod : USINT := TIME_UP_DOWN;
    END_STRUCT
END_TYPE

// BODAS_RC18_12_40/Application/02 EasyConfig/DSM_easyConfig/Structure/DFC_bds_NoDeb0x80a4
{attribute 'external_name' := 'cmp_rts_DFC_bds_NoDeb0x80a4'}
TYPE DFC_bds_NoDeb0x80a4 : STRUCT
        DTC            : UDINT := 16#80A400;
        DFCid          : UINT  := 171;
        debounceMethod : USINT := TIME_UP_DOWN;
    END_STRUCT
END_TYPE

// BODAS_RC18_12_40/Application/02 EasyConfig/DSM_easyConfig/Structure/DFC_bds_NoDeb0x80a5
{attribute 'external_name' := 'cmp_rts_DFC_bds_NoDeb0x80a5'}
TYPE DFC_bds_NoDeb0x80a5 : STRUCT
        DTC            : UDINT := 16#80A500;
        DFCid          : UINT  := 172;
        debounceMethod : USINT := TIME_UP_DOWN;
    END_STRUCT
END_TYPE

// BODAS_RC18_12_40/Application/02 EasyConfig/DSM_easyConfig/Structure/DFC_bds_NoDeb0x80a6
{attribute 'external_name' := 'cmp_rts_DFC_bds_NoDeb0x80a6'}
TYPE DFC_bds_NoDeb0x80a6 : STRUCT
        DTC            : UDINT := 16#80A600;
        DFCid          : UINT  := 173;
        debounceMethod : USINT := TIME_UP_DOWN;
    END_STRUCT
END_TYPE

// BODAS_RC18_12_40/Application/02 EasyConfig/DSM_easyConfig/Structure/DFC_bds_NoDeb0x80a7
{attribute 'external_name' := 'cmp_rts_DFC_bds_NoDeb0x80a7'}
TYPE DFC_bds_NoDeb0x80a7 : STRUCT
        DTC            : UDINT := 16#80A700;
        DFCid          : UINT  := 174;
        debounceMethod : USINT := TIME_UP_DOWN;
    END_STRUCT
END_TYPE

// BODAS_RC18_12_40/Application/02 EasyConfig/DSM_easyConfig/Structure/DFC_bds_NoDeb0x80a8
{attribute 'external_name' := 'cmp_rts_DFC_bds_NoDeb0x80a8'}
TYPE DFC_bds_NoDeb0x80a8 : STRUCT
        DTC            : UDINT := 16#80A800;
        DFCid          : UINT  := 175;
        debounceMethod : USINT := TIME_UP_DOWN;
    END_STRUCT
END_TYPE

// BODAS_RC18_12_40/Application/02 EasyConfig/DSM_easyConfig/Structure/DFC_bds_NoDeb0x80a9
{attribute 'external_name' := 'cmp_rts_DFC_bds_NoDeb0x80a9'}
TYPE DFC_bds_NoDeb0x80a9 : STRUCT
        DTC            : UDINT := 16#80A900;
        DFCid          : UINT  := 176;
        debounceMethod : USINT := TIME_UP_DOWN;
    END_STRUCT
END_TYPE

// BODAS_RC18_12_40/Application/02 EasyConfig/DSM_easyConfig/Structure/DFC_bds_NoDeb0x80aa
{attribute 'external_name' := 'cmp_rts_DFC_bds_NoDeb0x80aa'}
TYPE DFC_bds_NoDeb0x80aa : STRUCT
        DTC            : UDINT := 16#80AA00;
        DFCid          : UINT  := 177;
        debounceMethod : USINT := TIME_UP_DOWN;
    END_STRUCT
END_TYPE

// BODAS_RC18_12_40/Application/02 EasyConfig/DSM_easyConfig/Structure/DFC_bds_NoDeb0x80ab
{attribute 'external_name' := 'cmp_rts_DFC_bds_NoDeb0x80ab'}
TYPE DFC_bds_NoDeb0x80ab : STRUCT
        DTC            : UDINT := 16#80AB00;
        DFCid          : UINT  := 178;
        debounceMethod : USINT := TIME_UP_DOWN;
    END_STRUCT
END_TYPE

// BODAS_RC18_12_40/Application/02 EasyConfig/DSM_easyConfig/Structure/DFC_bds_NoDeb0x80ac
{attribute 'external_name' := 'cmp_rts_DFC_bds_NoDeb0x80ac'}
TYPE DFC_bds_NoDeb0x80ac : STRUCT
        DTC            : UDINT := 16#80AC00;
        DFCid          : UINT  := 179;
        debounceMethod : USINT := TIME_UP_DOWN;
    END_STRUCT
END_TYPE

// BODAS_RC18_12_40/Application/02 EasyConfig/DSM_easyConfig/Structure/DFC_bds_NoDeb0x80ad
{attribute 'external_name' := 'cmp_rts_DFC_bds_NoDeb0x80ad'}
TYPE DFC_bds_NoDeb0x80ad : STRUCT
        DTC            : UDINT := 16#80AD00;
        DFCid          : UINT  := 180;
        debounceMethod : USINT := TIME_UP_DOWN;
    END_STRUCT
END_TYPE

// BODAS_RC18_12_40/Application/02 EasyConfig/DSM_easyConfig/Structure/DFC_bds_NoDeb0x80ae
{attribute 'external_name' := 'cmp_rts_DFC_bds_NoDeb0x80ae'}
TYPE DFC_bds_NoDeb0x80ae : STRUCT
        DTC            : UDINT := 16#80AE00;
        DFCid          : UINT  := 181;
        debounceMethod : USINT := TIME_UP_DOWN;
    END_STRUCT
END_TYPE

// BODAS_RC18_12_40/Application/02 EasyConfig/DSM_easyConfig/Structure/DFC_bds_NoDeb0x80af
{attribute 'external_name' := 'cmp_rts_DFC_bds_NoDeb0x80af'}
TYPE DFC_bds_NoDeb0x80af : STRUCT
        DTC            : UDINT := 16#80AF00;
        DFCid          : UINT  := 182;
        debounceMethod : USINT := TIME_UP_DOWN;
    END_STRUCT
END_TYPE

// BODAS_RC18_12_40/Application/02 EasyConfig/DSM_easyConfig/Structure/DFC_bds_NoDeb0x80b0
{attribute 'external_name' := 'cmp_rts_DFC_bds_NoDeb0x80b0'}
TYPE DFC_bds_NoDeb0x80b0 : STRUCT
        DTC            : UDINT := 16#80B000;
        DFCid          : UINT  := 183;
        debounceMethod : USINT := TIME_UP_DOWN;
    END_STRUCT
END_TYPE

// BODAS_RC18_12_40/Application/02 EasyConfig/DSM_easyConfig/Structure/DFC_bds_NoDeb0x80b1
{attribute 'external_name' := 'cmp_rts_DFC_bds_NoDeb0x80b1'}
TYPE DFC_bds_NoDeb0x80b1 : STRUCT
        DTC            : UDINT := 16#80B100;
        DFCid          : UINT  := 184;
        debounceMethod : USINT := TIME_UP_DOWN;
    END_STRUCT
END_TYPE

// BODAS_RC18_12_40/Application/02 EasyConfig/DSM_easyConfig/Structure/DFC_bds_NoDeb0x80b2
{attribute 'external_name' := 'cmp_rts_DFC_bds_NoDeb0x80b2'}
TYPE DFC_bds_NoDeb0x80b2 : STRUCT
        DTC            : UDINT := 16#80B200;
        DFCid          : UINT  := 185;
        debounceMethod : USINT := TIME_UP_DOWN;
    END_STRUCT
END_TYPE

// BODAS_RC18_12_40/Application/02 EasyConfig/DSM_easyConfig/Structure/DFC_bds_NoDeb0x80b3
{attribute 'external_name' := 'cmp_rts_DFC_bds_NoDeb0x80b3'}
TYPE DFC_bds_NoDeb0x80b3 : STRUCT
        DTC            : UDINT := 16#80B300;
        DFCid          : UINT  := 186;
        debounceMethod : USINT := TIME_UP_DOWN;
    END_STRUCT
END_TYPE

// BODAS_RC18_12_40/Application/02 EasyConfig/DSM_easyConfig/Structure/DFC_bds_NoDeb0x80b4
{attribute 'external_name' := 'cmp_rts_DFC_bds_NoDeb0x80b4'}
TYPE DFC_bds_NoDeb0x80b4 : STRUCT
        DTC            : UDINT := 16#80B400;
        DFCid          : UINT  := 187;
        debounceMethod : USINT := TIME_UP_DOWN;
    END_STRUCT
END_TYPE

// BODAS_RC18_12_40/Application/02 EasyConfig/DSM_easyConfig/Structure/DFC_bds_NoDeb0x80b5
{attribute 'external_name' := 'cmp_rts_DFC_bds_NoDeb0x80b5'}
TYPE DFC_bds_NoDeb0x80b5 : STRUCT
        DTC            : UDINT := 16#80B500;
        DFCid          : UINT  := 188;
        debounceMethod : USINT := TIME_UP_DOWN;
    END_STRUCT
END_TYPE

// BODAS_RC18_12_40/Application/02 EasyConfig/DSM_easyConfig/Structure/DFC_bds_NoDeb0x80b6
{attribute 'external_name' := 'cmp_rts_DFC_bds_NoDeb0x80b6'}
TYPE DFC_bds_NoDeb0x80b6 : STRUCT
        DTC            : UDINT := 16#80B600;
        DFCid          : UINT  := 189;
        debounceMethod : USINT := TIME_UP_DOWN;
    END_STRUCT
END_TYPE

// BODAS_RC18_12_40/Application/02 EasyConfig/DSM_easyConfig/Structure/DFC_bds_NoDeb0x80b7
{attribute 'external_name' := 'cmp_rts_DFC_bds_NoDeb0x80b7'}
TYPE DFC_bds_NoDeb0x80b7 : STRUCT
        DTC            : UDINT := 16#80B700;
        DFCid          : UINT  := 190;
        debounceMethod : USINT := TIME_UP_DOWN;
    END_STRUCT
END_TYPE

// BODAS_RC18_12_40/Application/02 EasyConfig/DSM_easyConfig/Structure/DFC_bds_NoDeb0x80b8
{attribute 'external_name' := 'cmp_rts_DFC_bds_NoDeb0x80b8'}
TYPE DFC_bds_NoDeb0x80b8 : STRUCT
        DTC            : UDINT := 16#80B800;
        DFCid          : UINT  := 191;
        debounceMethod : USINT := TIME_UP_DOWN;
    END_STRUCT
END_TYPE

// BODAS_RC18_12_40/Application/02 EasyConfig/DSM_easyConfig/Structure/DFC_bds_NoDeb0x80b9
{attribute 'external_name' := 'cmp_rts_DFC_bds_NoDeb0x80b9'}
TYPE DFC_bds_NoDeb0x80b9 : STRUCT
        DTC            : UDINT := 16#80B900;
        DFCid          : UINT  := 192;
        debounceMethod : USINT := TIME_UP_DOWN;
    END_STRUCT
END_TYPE

// BODAS_RC18_12_40/Application/02 EasyConfig/DSM_easyConfig/Structure/DFC_bds_NoDeb0x80ba
{attribute 'external_name' := 'cmp_rts_DFC_bds_NoDeb0x80ba'}
TYPE DFC_bds_NoDeb0x80ba : STRUCT
        DTC            : UDINT := 16#80BA00;
        DFCid          : UINT  := 193;
        debounceMethod : USINT := TIME_UP_DOWN;
    END_STRUCT
END_TYPE

// BODAS_RC18_12_40/Application/02 EasyConfig/DSM_easyConfig/Structure/DFC_bds_NoDeb0x80bb
{attribute 'external_name' := 'cmp_rts_DFC_bds_NoDeb0x80bb'}
TYPE DFC_bds_NoDeb0x80bb : STRUCT
        DTC            : UDINT := 16#80BB00;
        DFCid          : UINT  := 194;
        debounceMethod : USINT := TIME_UP_DOWN;
    END_STRUCT
END_TYPE

// BODAS_RC18_12_40/Application/02 EasyConfig/DSM_easyConfig/Structure/DFC_bds_NoDeb0x80bc
{attribute 'external_name' := 'cmp_rts_DFC_bds_NoDeb0x80bc'}
TYPE DFC_bds_NoDeb0x80bc : STRUCT
        DTC            : UDINT := 16#80BC00;
        DFCid          : UINT  := 195;
        debounceMethod : USINT := TIME_UP_DOWN;
    END_STRUCT
END_TYPE

// BODAS_RC18_12_40/Application/02 EasyConfig/DSM_easyConfig/Structure/DFC_bds_NoDeb0x80bd
{attribute 'external_name' := 'cmp_rts_DFC_bds_NoDeb0x80bd'}
TYPE DFC_bds_NoDeb0x80bd : STRUCT
        DTC            : UDINT := 16#80BD00;
        DFCid          : UINT  := 196;
        debounceMethod : USINT := TIME_UP_DOWN;
    END_STRUCT
END_TYPE

// BODAS_RC18_12_40/Application/02 EasyConfig/DSM_easyConfig/Structure/DFC_bds_NoDeb0x80be
{attribute 'external_name' := 'cmp_rts_DFC_bds_NoDeb0x80be'}
TYPE DFC_bds_NoDeb0x80be : STRUCT
        DTC            : UDINT := 16#80BE00;
        DFCid          : UINT  := 197;
        debounceMethod : USINT := TIME_UP_DOWN;
    END_STRUCT
END_TYPE

// BODAS_RC18_12_40/Application/02 EasyConfig/DSM_easyConfig/Structure/DFC_bds_NoDeb0x80bf
{attribute 'external_name' := 'cmp_rts_DFC_bds_NoDeb0x80bf'}
TYPE DFC_bds_NoDeb0x80bf : STRUCT
        DTC            : UDINT := 16#80BF00;
        DFCid          : UINT  := 198;
        debounceMethod : USINT := TIME_UP_DOWN;
    END_STRUCT
END_TYPE

// BODAS_RC18_12_40/Application/02 EasyConfig/DSM_easyConfig/Structure/DFC_bds_NoDeb0x80c0
{attribute 'external_name' := 'cmp_rts_DFC_bds_NoDeb0x80c0'}
TYPE DFC_bds_NoDeb0x80c0 : STRUCT
        DTC            : UDINT := 16#80C000;
        DFCid          : UINT  := 199;
        debounceMethod : USINT := TIME_UP_DOWN;
    END_STRUCT
END_TYPE

// BODAS_RC18_12_40/Application/02 EasyConfig/DSM_easyConfig/Structure/DFC_bds_NoDeb0x80c1
{attribute 'external_name' := 'cmp_rts_DFC_bds_NoDeb0x80c1'}
TYPE DFC_bds_NoDeb0x80c1 : STRUCT
        DTC            : UDINT := 16#80C100;
        DFCid          : UINT  := 200;
        debounceMethod : USINT := TIME_UP_DOWN;
    END_STRUCT
END_TYPE

// BODAS_RC18_12_40/Application/02 EasyConfig/DSM_easyConfig/Structure/DFC_bds_NoDeb0x80c2
{attribute 'external_name' := 'cmp_rts_DFC_bds_NoDeb0x80c2'}
TYPE DFC_bds_NoDeb0x80c2 : STRUCT
        DTC            : UDINT := 16#80C200;
        DFCid          : UINT  := 201;
        debounceMethod : USINT := TIME_UP_DOWN;
    END_STRUCT
END_TYPE

// BODAS_RC18_12_40/Application/02 EasyConfig/DSM_easyConfig/Structure/DFC_bds_NoDeb0x80c3
{attribute 'external_name' := 'cmp_rts_DFC_bds_NoDeb0x80c3'}
TYPE DFC_bds_NoDeb0x80c3 : STRUCT
        DTC            : UDINT := 16#80C300;
        DFCid          : UINT  := 202;
        debounceMethod : USINT := TIME_UP_DOWN;
    END_STRUCT
END_TYPE

// BODAS_RC18_12_40/Application/02 EasyConfig/DSM_easyConfig/Structure/DFC_bds_NoDeb0x80c4
{attribute 'external_name' := 'cmp_rts_DFC_bds_NoDeb0x80c4'}
TYPE DFC_bds_NoDeb0x80c4 : STRUCT
        DTC            : UDINT := 16#80C400;
        DFCid          : UINT  := 203;
        debounceMethod : USINT := TIME_UP_DOWN;
    END_STRUCT
END_TYPE

// BODAS_RC18_12_40/Application/02 EasyConfig/DSM_easyConfig/Structure/DFC_bds_NoDeb0x80c5
{attribute 'external_name' := 'cmp_rts_DFC_bds_NoDeb0x80c5'}
TYPE DFC_bds_NoDeb0x80c5 : STRUCT
        DTC            : UDINT := 16#80C500;
        DFCid          : UINT  := 204;
        debounceMethod : USINT := TIME_UP_DOWN;
    END_STRUCT
END_TYPE

// BODAS_RC18_12_40/Application/02 EasyConfig/DSM_easyConfig/Structure/DFC_bds_NoDeb0x80c6
{attribute 'external_name' := 'cmp_rts_DFC_bds_NoDeb0x80c6'}
TYPE DFC_bds_NoDeb0x80c6 : STRUCT
        DTC            : UDINT := 16#80C600;
        DFCid          : UINT  := 205;
        debounceMethod : USINT := TIME_UP_DOWN;
    END_STRUCT
END_TYPE

// BODAS_RC18_12_40/Application/02 EasyConfig/DSM_easyConfig/Structure/DFC_bds_NoDeb0x80c7
{attribute 'external_name' := 'cmp_rts_DFC_bds_NoDeb0x80c7'}
TYPE DFC_bds_NoDeb0x80c7 : STRUCT
        DTC            : UDINT := 16#80C700;
        DFCid          : UINT  := 1;
        debounceMethod : USINT := TIME_IN_ROW;
    END_STRUCT
END_TYPE

// BODAS_RC18_12_40/Application/02 EasyConfig/DSM_easyConfig/Structure/DFC_bds_NoDeb0x80c8
{attribute 'external_name' := 'cmp_rts_DFC_bds_NoDeb0x80c8'}
TYPE DFC_bds_NoDeb0x80c8 : STRUCT
        DTC            : UDINT := 16#80C800;
        DFCid          : UINT  := 2;
        debounceMethod : USINT := TIME_IN_ROW;
    END_STRUCT
END_TYPE

// BODAS_RC18_12_40/Application/02 EasyConfig/DSM_easyConfig/Structure/DFC_bds_NoDeb0x80c9
{attribute 'external_name' := 'cmp_rts_DFC_bds_NoDeb0x80c9'}
TYPE DFC_bds_NoDeb0x80c9 : STRUCT
        DTC            : UDINT := 16#80C900;
        DFCid          : UINT  := 3;
        debounceMethod : USINT := TIME_IN_ROW;
    END_STRUCT
END_TYPE

// BODAS_RC18_12_40/Application/02 EasyConfig/DSM_easyConfig/Structure/DFC_bds_NoDeb0x80ca
{attribute 'external_name' := 'cmp_rts_DFC_bds_NoDeb0x80ca'}
TYPE DFC_bds_NoDeb0x80ca : STRUCT
        DTC            : UDINT := 16#80CA00;
        DFCid          : UINT  := 4;
        debounceMethod : USINT := TIME_IN_ROW;
    END_STRUCT
END_TYPE

// BODAS_RC18_12_40/Application/02 EasyConfig/DSM_easyConfig/Structure/DFC_bds_NoDeb0x80cb
{attribute 'external_name' := 'cmp_rts_DFC_bds_NoDeb0x80cb'}
TYPE DFC_bds_NoDeb0x80cb : STRUCT
        DTC            : UDINT := 16#80CB00;
        DFCid          : UINT  := 5;
        debounceMethod : USINT := TIME_IN_ROW;
    END_STRUCT
END_TYPE

// BODAS_RC18_12_40/Application/02 EasyConfig/DSM_easyConfig/Structure/DFC_bds_NoDeb0x80cc
{attribute 'external_name' := 'cmp_rts_DFC_bds_NoDeb0x80cc'}
TYPE DFC_bds_NoDeb0x80cc : STRUCT
        DTC            : UDINT := 16#80CC00;
        DFCid          : UINT  := 6;
        debounceMethod : USINT := TIME_IN_ROW;
    END_STRUCT
END_TYPE

// BODAS_RC18_12_40/Application/02 EasyConfig/DSM_easyConfig/Structure/DFC_bds_NoDeb0x80cd
{attribute 'external_name' := 'cmp_rts_DFC_bds_NoDeb0x80cd'}
TYPE DFC_bds_NoDeb0x80cd : STRUCT
        DTC            : UDINT := 16#80CD00;
        DFCid          : UINT  := 7;
        debounceMethod : USINT := TIME_IN_ROW;
    END_STRUCT
END_TYPE

// BODAS_RC18_12_40/Application/02 EasyConfig/DSM_easyConfig/Structure/DFC_bds_NoDeb0x80ce
{attribute 'external_name' := 'cmp_rts_DFC_bds_NoDeb0x80ce'}
TYPE DFC_bds_NoDeb0x80ce : STRUCT
        DTC            : UDINT := 16#80CE00;
        DFCid          : UINT  := 8;
        debounceMethod : USINT := TIME_IN_ROW;
    END_STRUCT
END_TYPE

// BODAS_RC18_12_40/Application/02 EasyConfig/DSM_easyConfig/Structure/DFC_bds_NoDeb0x80cf
{attribute 'external_name' := 'cmp_rts_DFC_bds_NoDeb0x80cf'}
TYPE DFC_bds_NoDeb0x80cf : STRUCT
        DTC            : UDINT := 16#80CF00;
        DFCid          : UINT  := 9;
        debounceMethod : USINT := TIME_IN_ROW;
    END_STRUCT
END_TYPE

// BODAS_RC18_12_40/Application/02 EasyConfig/DSM_easyConfig/Structure/DFC_bds_NoDeb0x80d0
{attribute 'external_name' := 'cmp_rts_DFC_bds_NoDeb0x80d0'}
TYPE DFC_bds_NoDeb0x80d0 : STRUCT
        DTC            : UDINT := 16#80D000;
        DFCid          : UINT  := 10;
        debounceMethod : USINT := TIME_IN_ROW;
    END_STRUCT
END_TYPE

// BODAS_RC18_12_40/Application/02 EasyConfig/DSM_easyConfig/Structure/DFC_bds_NoDeb0x80d1
{attribute 'external_name' := 'cmp_rts_DFC_bds_NoDeb0x80d1'}
TYPE DFC_bds_NoDeb0x80d1 : STRUCT
        DTC            : UDINT := 16#80D100;
        DFCid          : UINT  := 11;
        debounceMethod : USINT := TIME_IN_ROW;
    END_STRUCT
END_TYPE

// BODAS_RC18_12_40/Application/02 EasyConfig/DSM_easyConfig/Structure/DFC_bds_NoDeb0x80d2
{attribute 'external_name' := 'cmp_rts_DFC_bds_NoDeb0x80d2'}
TYPE DFC_bds_NoDeb0x80d2 : STRUCT
        DTC            : UDINT := 16#80D200;
        DFCid          : UINT  := 12;
        debounceMethod : USINT := TIME_IN_ROW;
    END_STRUCT
END_TYPE

// BODAS_RC18_12_40/Application/02 EasyConfig/DSM_easyConfig/Structure/DFC_bds_NoDeb0x80d3
{attribute 'external_name' := 'cmp_rts_DFC_bds_NoDeb0x80d3'}
TYPE DFC_bds_NoDeb0x80d3 : STRUCT
        DTC            : UDINT := 16#80D300;
        DFCid          : UINT  := 13;
        debounceMethod : USINT := TIME_IN_ROW;
    END_STRUCT
END_TYPE

// BODAS_RC18_12_40/Application/02 EasyConfig/DSM_easyConfig/Structure/DFC_bds_NoDeb0x80d4
{attribute 'external_name' := 'cmp_rts_DFC_bds_NoDeb0x80d4'}
TYPE DFC_bds_NoDeb0x80d4 : STRUCT
        DTC            : UDINT := 16#80D400;
        DFCid          : UINT  := 14;
        debounceMethod : USINT := TIME_IN_ROW;
    END_STRUCT
END_TYPE

// BODAS_RC18_12_40/Application/02 EasyConfig/DSM_easyConfig/Structure/DFC_bds_NoDeb0x80d5
{attribute 'external_name' := 'cmp_rts_DFC_bds_NoDeb0x80d5'}
TYPE DFC_bds_NoDeb0x80d5 : STRUCT
        DTC            : UDINT := 16#80D500;
        DFCid          : UINT  := 15;
        debounceMethod : USINT := TIME_IN_ROW;
    END_STRUCT
END_TYPE

// BODAS_RC18_12_40/Application/02 EasyConfig/DSM_easyConfig/Structure/DFC_bds_NoDeb0x80d6
{attribute 'external_name' := 'cmp_rts_DFC_bds_NoDeb0x80d6'}
TYPE DFC_bds_NoDeb0x80d6 : STRUCT
        DTC            : UDINT := 16#80D600;
        DFCid          : UINT  := 16;
        debounceMethod : USINT := TIME_IN_ROW;
    END_STRUCT
END_TYPE

// BODAS_RC18_12_40/Application/02 EasyConfig/DSM_easyConfig/Structure/DFC_bds_NoDeb0x80d7
{attribute 'external_name' := 'cmp_rts_DFC_bds_NoDeb0x80d7'}
TYPE DFC_bds_NoDeb0x80d7 : STRUCT
        DTC            : UDINT := 16#80D700;
        DFCid          : UINT  := 17;
        debounceMethod : USINT := TIME_IN_ROW;
    END_STRUCT
END_TYPE

// BODAS_RC18_12_40/Application/02 EasyConfig/DSM_easyConfig/Structure/DFC_bds_NoDeb0x80d8
{attribute 'external_name' := 'cmp_rts_DFC_bds_NoDeb0x80d8'}
TYPE DFC_bds_NoDeb0x80d8 : STRUCT
        DTC            : UDINT := 16#80D800;
        DFCid          : UINT  := 18;
        debounceMethod : USINT := TIME_IN_ROW;
    END_STRUCT
END_TYPE

// BODAS_RC18_12_40/Application/02 EasyConfig/DSM_easyConfig/Structure/DFC_bds_NoDeb0x80d9
{attribute 'external_name' := 'cmp_rts_DFC_bds_NoDeb0x80d9'}
TYPE DFC_bds_NoDeb0x80d9 : STRUCT
        DTC            : UDINT := 16#80D900;
        DFCid          : UINT  := 19;
        debounceMethod : USINT := TIME_IN_ROW;
    END_STRUCT
END_TYPE

// BODAS_RC18_12_40/Application/02 EasyConfig/DSM_easyConfig/Structure/DFC_bds_NoDeb0x80da
{attribute 'external_name' := 'cmp_rts_DFC_bds_NoDeb0x80da'}
TYPE DFC_bds_NoDeb0x80da : STRUCT
        DTC            : UDINT := 16#80DA00;
        DFCid          : UINT  := 20;
        debounceMethod : USINT := TIME_IN_ROW;
    END_STRUCT
END_TYPE

// BODAS_RC18_12_40/Application/02 EasyConfig/DSM_easyConfig/Structure/DFC_bds_NoDeb0x80db
{attribute 'external_name' := 'cmp_rts_DFC_bds_NoDeb0x80db'}
TYPE DFC_bds_NoDeb0x80db : STRUCT
        DTC            : UDINT := 16#80DB00;
        DFCid          : UINT  := 21;
        debounceMethod : USINT := TIME_IN_ROW;
    END_STRUCT
END_TYPE

// BODAS_RC18_12_40/Application/02 EasyConfig/DSM_easyConfig/Structure/DFC_bds_NoDeb0x80dc
{attribute 'external_name' := 'cmp_rts_DFC_bds_NoDeb0x80dc'}
TYPE DFC_bds_NoDeb0x80dc : STRUCT
        DTC            : UDINT := 16#80DC00;
        DFCid          : UINT  := 22;
        debounceMethod : USINT := TIME_IN_ROW;
    END_STRUCT
END_TYPE

// BODAS_RC18_12_40/Application/02 EasyConfig/DSM_easyConfig/Structure/DFC_bds_NoDeb0x80dd
{attribute 'external_name' := 'cmp_rts_DFC_bds_NoDeb0x80dd'}
TYPE DFC_bds_NoDeb0x80dd : STRUCT
        DTC            : UDINT := 16#80DD00;
        DFCid          : UINT  := 23;
        debounceMethod : USINT := TIME_IN_ROW;
    END_STRUCT
END_TYPE

// BODAS_RC18_12_40/Application/02 EasyConfig/DSM_easyConfig/Structure/DFC_bds_NoDeb0x80de
{attribute 'external_name' := 'cmp_rts_DFC_bds_NoDeb0x80de'}
TYPE DFC_bds_NoDeb0x80de : STRUCT
        DTC            : UDINT := 16#80DE00;
        DFCid          : UINT  := 24;
        debounceMethod : USINT := TIME_IN_ROW;
    END_STRUCT
END_TYPE

// BODAS_RC18_12_40/Application/02 EasyConfig/DSM_easyConfig/Structure/DFC_bds_NoDeb0x80df
{attribute 'external_name' := 'cmp_rts_DFC_bds_NoDeb0x80df'}
TYPE DFC_bds_NoDeb0x80df : STRUCT
        DTC            : UDINT := 16#80DF00;
        DFCid          : UINT  := 25;
        debounceMethod : USINT := TIME_IN_ROW;
    END_STRUCT
END_TYPE

// BODAS_RC18_12_40/Application/02 EasyConfig/DSM_easyConfig/Structure/DFC_bds_NoDeb0x80e0
{attribute 'external_name' := 'cmp_rts_DFC_bds_NoDeb0x80e0'}
TYPE DFC_bds_NoDeb0x80e0 : STRUCT
        DTC            : UDINT := 16#80E000;
        DFCid          : UINT  := 26;
        debounceMethod : USINT := TIME_IN_ROW;
    END_STRUCT
END_TYPE

// BODAS_RC18_12_40/Application/02 EasyConfig/DSM_easyConfig/Structure/DFC_bds_NoDeb0x80e1
{attribute 'external_name' := 'cmp_rts_DFC_bds_NoDeb0x80e1'}
TYPE DFC_bds_NoDeb0x80e1 : STRUCT
        DTC            : UDINT := 16#80E100;
        DFCid          : UINT  := 27;
        debounceMethod : USINT := TIME_IN_ROW;
    END_STRUCT
END_TYPE

